// TIA Portal V20 export
FUNCTION_BLOCK "Sequence_10_GaugeRnR"   // FB32857, LAD
TITLE = Sequence
// Sequence template programmend in ladder logic
// stored: IsIECCheckEnabled true, MemoryReserve 100, Namespace Unit1.Em5, SetENOAutomatically true
   VAR_INPUT
      unitStatus { ExternalAccessible := 'False'; ExternalVisible := 'False'; ExternalWritable := 'False'} : "LAF_typeUnitStatus";
   END_VAR
   VAR
      instSequenceLADControl { ExternalWritable := 'False'} : "LAF_ControlLadSequence";
      instSequenceLADStatus { ExternalWritable := 'False'} : "LAF_StatusLadSequence";
      statTonTime { ExternalAccessible := 'False'; ExternalVisible := 'False'; ExternalWritable := 'False'} : Array[0..9999] of TON_TIME;
   END_VAR
   VAR_TEMP
      tempCustomerAction : Bool;   // Placeholder for possible actions
      tempDo_nothing_and_wait_for_init : Bool;   // Placeholder for doing nothing
      tempSafeStateCondition : Bool;   // Temp Condition for the equipment module to be in a safe state
   END_VAR
   VAR CONSTANT
      delayTime : Time := T#500ms;
      STEP_IDLE : DInt := 1;
      JOB_1_STEP_01 : DInt := 101;
      JOB_1_STEP_10 : DInt := 110;
      JOB_1_STEP_20 : DInt := 120;
      JOB_1_STEP_30 : DInt := 130;
      JOB_1_STEP_40 : DInt := 140;
      JOB_1_STEP_50 : DInt := 150;
      JOB_1_STEP_60 : DInt := 160;
      JOB_1_STEP_70 : DInt := 170;
      JOB_1_STEP_80 : DInt := 180;
      JOB_1_STEP_90 : DInt := 190;
      JOB_2_STEP_01 : DInt := 201;
      JOB_2_STEP_10 : DInt := 210;
      JOB_2_STEP_20 : DInt := 220;
      JOB_2_STEP_30 : DInt := 230;
      JOB_2_STEP_40 : DInt := 240;
      JOB_2_STEP_41 : DInt := 241;
      JOB_2_STEP_80 : DInt := 280;
      JOB_2_STEP_81 : DInt := 281;
      JOB_2_STEP_90 : DInt := 290;
      JOB_3_STEP_01 : DInt := 301;
      JOB_3_STEP_10 : DInt := 310;
      JOB_3_STEP_20 : DInt := 320;
      JOB_3_STEP_30 : DInt := 330;
      JOB_3_STEP_40 : DInt := 340;
      JOB_3_STEP_50 : DInt := 350;
      JOB_3_STEP_80 : DInt := 380;
      JOB_3_STEP_81 : DInt := 381;
      JOB_3_STEP_82 : DInt := 382;
      JOB_3_STEP_90 : DInt := 390;
      JOB_4_STEP_01 : DInt := 401;
      JOB_4_STEP_10 : DInt := 410;
      JOB_4_STEP_20 : DInt := 420;
      JOB_4_STEP_30 : DInt := 430;
      JOB_4_STEP_40 : DInt := 440;
      JOB_4_STEP_50 : DInt := 450;
      JOB_4_STEP_60 : DInt := 460;
      JOB_4_STEP_70 : DInt := 470;
      JOB_4_STEP_80 : DInt := 480;
      JOB_4_STEP_81 : DInt := 481;
      JOB_4_STEP_90 : DInt := 490;
      JOB_5_STEP_01 : DInt := 501;
      JOB_5_STEP_10 : DInt := 510;
      JOB_5_STEP_20 : DInt := 520;
      JOB_5_STEP_30 : DInt := 530;
      JOB_5_STEP_40 : DInt := 540;
      JOB_5_STEP_50 : DInt := 550;
      JOB_5_STEP_60 : DInt := 560;
      JOB_5_STEP_70 : DInt := 570;
      JOB_5_STEP_80 : DInt := 580;
      JOB_5_STEP_81 : DInt := 581;
      JOB_5_STEP_90 : DInt := 590;
      JOB_6_STEP_01 : DInt := 601;
      JOB_6_STEP_10 : DInt := 610;
      JOB_6_STEP_20 : DInt := 620;
      JOB_6_STEP_30 : DInt := 630;
      JOB_6_STEP_40 : DInt := 640;
      JOB_6_STEP_50 : DInt := 650;
      JOB_6_STEP_60 : DInt := 660;
      JOB_6_STEP_70 : DInt := 670;
      JOB_6_STEP_80 : DInt := 680;
      JOB_6_STEP_81 : DInt := 681;
      JOB_6_STEP_82 : DInt := 682;
      JOB_6_STEP_90 : DInt := 690;
      JOB_7_STEP_01 : DInt := 701;
      JOB_7_STEP_10 : DInt := 710;
      JOB_7_STEP_20 : DInt := 720;
      JOB_7_STEP_30 : DInt := 730;
      JOB_7_STEP_40 : DInt := 740;
      JOB_7_STEP_50 : DInt := 750;
      JOB_7_STEP_60 : DInt := 760;
      JOB_7_STEP_70 : DInt := 770;
      JOB_7_STEP_80 : DInt := 780;
      JOB_7_STEP_81 : DInt := 781;
      JOB_7_STEP_82 : DInt := 782;
      JOB_7_STEP_90 : DInt := 790;
      JOB_8_STEP_01 : DInt := 801;
      JOB_8_STEP_10 : DInt := 810;
      JOB_8_STEP_20 : DInt := 820;
      JOB_8_STEP_30 : DInt := 830;
      JOB_8_STEP_31 : DInt := 831;
      JOB_8_STEP_40 : DInt := 840;
      JOB_8_STEP_50 : DInt := 850;
      JOB_8_STEP_80 : DInt := 880;
      JOB_8_STEP_81 : DInt := 881;
      JOB_8_STEP_90 : DInt := 890;
      JOB_9_STEP_01 : DInt := 901;
      JOB_9_STEP_10 : DInt := 910;
      JOB_9_STEP_20 : DInt := 920;
      JOB_9_STEP_30 : DInt := 930;
      JOB_9_STEP_40 : DInt := 940;
      JOB_9_STEP_80 : DInt := 980;
      JOB_9_STEP_81 : DInt := 981;
      JOB_9_STEP_90 : DInt := 990;
      STEP_IMMEDIATE_STOP : DInt := 9001;   // Step executed when an immediate stop command is triggered for the sequence (i.e. when unit is in state aborting)
      TO_DO_INSERT_ACTIONS_HERE : Bool := TRUE;   // Template : Add actions
      TO_DO_INSERT_CONDITION_FOR_TRANSITION_HERE : Bool := TRUE;   // Template : Add conditions
   END_VAR
   VAR_TEMP   // added for the SCL form of the ladder/FBD networks
      _w1 : Bool;
   END_VAR
BEGIN

REGION Network 1: BLOCK INFO HEADER
   // (company) / (C) Copyright (year)
   // ---------------------------------------------------------------------------------
   // Title:                             (Title of this block)
   // Comment/Function: (that is implemented in the block)
   // Library/Family:           (that the source is dedicated to)
   // Author:                        (department / person in charge / contact)
   // Target System:          (test system with FW version)
   // Engineering:              TIA Portal (SW version)
   // Restrictions:               (OB types, etc.)
   // Requirements:           (hardware, technological package, etc.)
   // ---------------------------------------------------------------------------------
   // Change log table:
   // Version          | Date             | Signature      | Expert in charge  | Changes applied ------------------------|----------------------|-------------------------|--------------------------------|-----------------------
   // 001.000.000 | yyyy-mm-dd | 0x00000000 | (name of expert) | First released version
END_REGION

REGION Network 2: DESCRIPTION
   // This is a template block provided by the Automation Framework. It can be used to create an own project.
   // The Block Info Header is prepared to put in your own data.
   // Description of the block could be added here and the docu created by Code2Docu.
END_REGION

REGION Network 3: ********************* CONTROL *************************
END_REGION

REGION Network 4: Sequence Control ("Enter your Sequins number here")
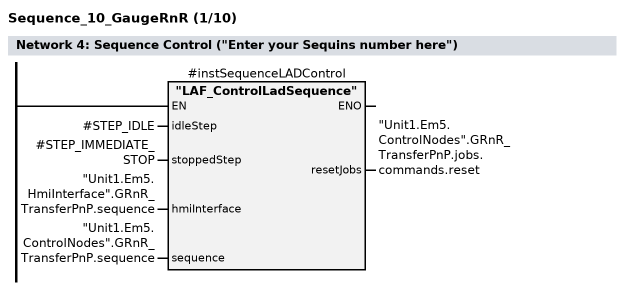
   RUNG wire#powerrail
      #instSequenceLADControl(idleStep := #STEP_IDLE, stoppedStep := #STEP_IMMEDIATE_STOP, hmiInterface := "Unit1.Em5.HmiInterface".GRnR_TransferPnP.sequence, sequence := "Unit1.Em5.ControlNodes".GRnR_TransferPnP.sequence, resetJobs => "Unit1.Em5.ControlNodes".GRnR_TransferPnP.jobs.commands.reset)
   END_RUNG
   // the same network as SCL:
   #instSequenceLADControl(idleStep := #STEP_IDLE,   // "LAF_ControlLadSequence"
                           stoppedStep := #STEP_IMMEDIATE_STOP,
                           hmiInterface := "Unit1.Em5.HmiInterface".GRnR_TransferPnP.sequence,
                           sequence := "Unit1.Em5.ControlNodes".GRnR_TransferPnP.sequence,
                           resetJobs => "Unit1.Em5.ControlNodes".GRnR_TransferPnP.jobs.commands.reset);
END_REGION

REGION Network 5: Step Idle
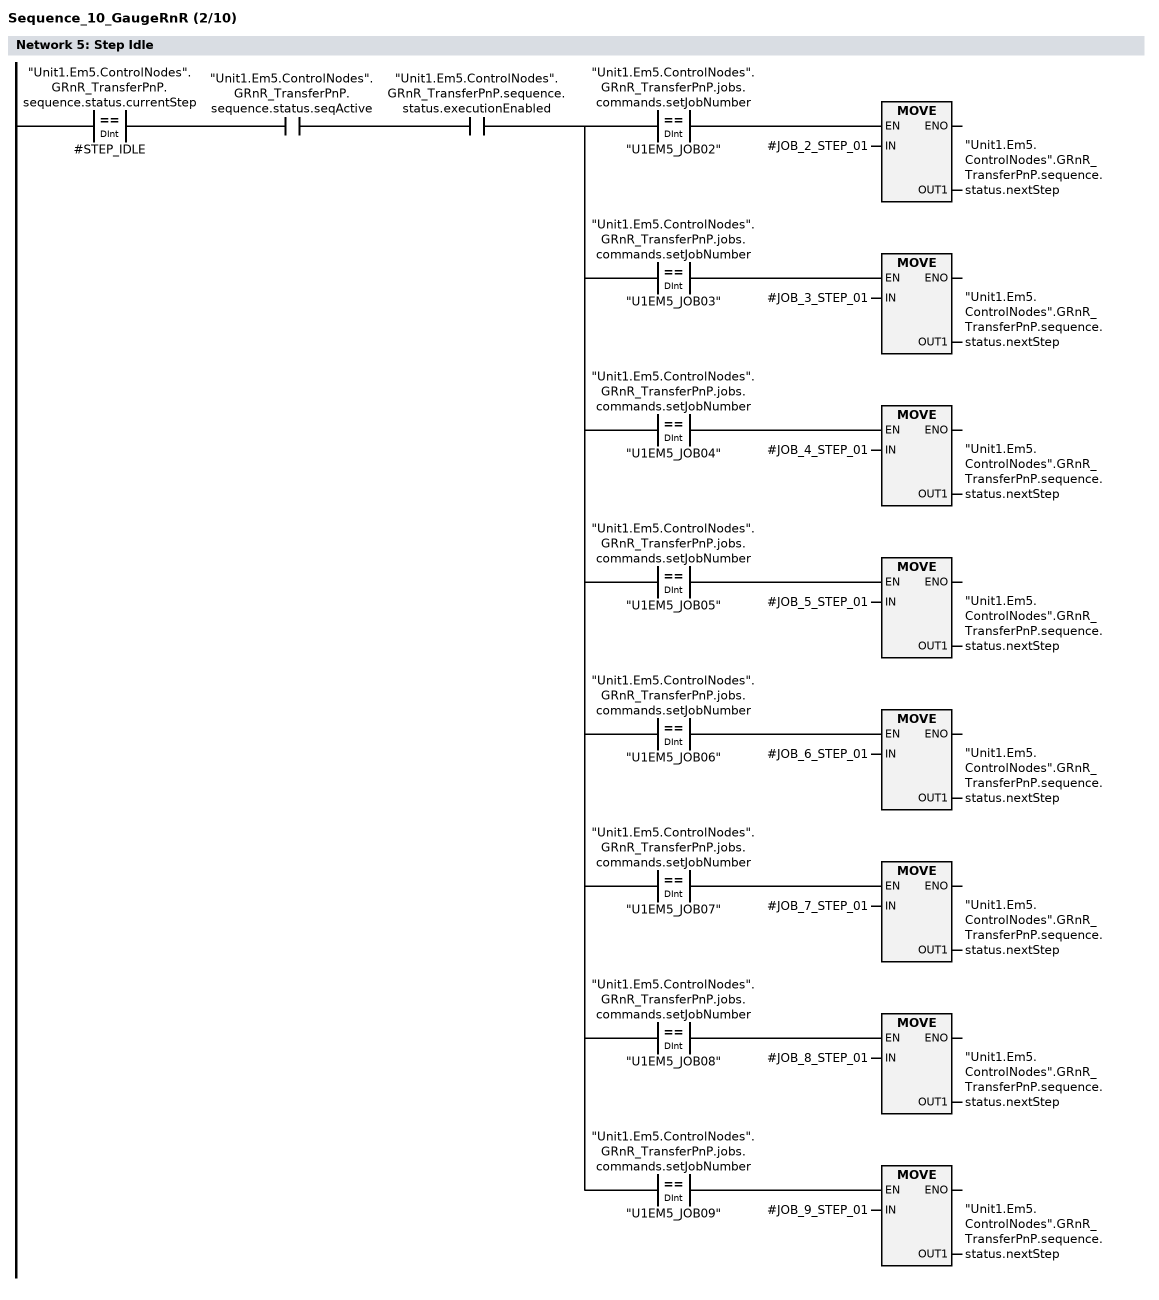
   RUNG wire#powerrail
      { S7_Templates := "SrcType := DInt" } EQ_Contact(in1 := "Unit1.Em5.ControlNodes".GRnR_TransferPnP.sequence.status.currentStep, in2 := #STEP_IDLE)
      Contact( "Unit1.Em5.ControlNodes".GRnR_TransferPnP.sequence.status.seqActive )
      Contact( "Unit1.Em5.ControlNodes".GRnR_TransferPnP.sequence.status.executionEnabled )
      wire#w1
      { S7_Templates := "SrcType := DInt" } EQ_Contact(in1 := "Unit1.Em5.ControlNodes".GRnR_TransferPnP.jobs.commands.setJobNumber, in2 := "U1EM5_JOB02")
      Move(in := #JOB_2_STEP_01, out1 => "Unit1.Em5.ControlNodes".GRnR_TransferPnP.sequence.status.nextStep)
   END_RUNG
   RUNG wire#w1
      { S7_Templates := "SrcType := DInt" } EQ_Contact(in1 := "Unit1.Em5.ControlNodes".GRnR_TransferPnP.jobs.commands.setJobNumber, in2 := "U1EM5_JOB03")
      Move(in := #JOB_3_STEP_01, out1 => "Unit1.Em5.ControlNodes".GRnR_TransferPnP.sequence.status.nextStep)
   END_RUNG
   RUNG wire#w1
      { S7_Templates := "SrcType := DInt" } EQ_Contact(in1 := "Unit1.Em5.ControlNodes".GRnR_TransferPnP.jobs.commands.setJobNumber, in2 := "U1EM5_JOB04")
      Move(in := #JOB_4_STEP_01, out1 => "Unit1.Em5.ControlNodes".GRnR_TransferPnP.sequence.status.nextStep)
   END_RUNG
   RUNG wire#w1
      { S7_Templates := "SrcType := DInt" } EQ_Contact(in1 := "Unit1.Em5.ControlNodes".GRnR_TransferPnP.jobs.commands.setJobNumber, in2 := "U1EM5_JOB05")
      Move(in := #JOB_5_STEP_01, out1 => "Unit1.Em5.ControlNodes".GRnR_TransferPnP.sequence.status.nextStep)
   END_RUNG
   RUNG wire#w1
      { S7_Templates := "SrcType := DInt" } EQ_Contact(in1 := "Unit1.Em5.ControlNodes".GRnR_TransferPnP.jobs.commands.setJobNumber, in2 := "U1EM5_JOB06")
      Move(in := #JOB_6_STEP_01, out1 => "Unit1.Em5.ControlNodes".GRnR_TransferPnP.sequence.status.nextStep)
   END_RUNG
   RUNG wire#w1
      { S7_Templates := "SrcType := DInt" } EQ_Contact(in1 := "Unit1.Em5.ControlNodes".GRnR_TransferPnP.jobs.commands.setJobNumber, in2 := "U1EM5_JOB07")
      Move(in := #JOB_7_STEP_01, out1 => "Unit1.Em5.ControlNodes".GRnR_TransferPnP.sequence.status.nextStep)
   END_RUNG
   RUNG wire#w1
      { S7_Templates := "SrcType := DInt" } EQ_Contact(in1 := "Unit1.Em5.ControlNodes".GRnR_TransferPnP.jobs.commands.setJobNumber, in2 := "U1EM5_JOB08")
      Move(in := #JOB_8_STEP_01, out1 => "Unit1.Em5.ControlNodes".GRnR_TransferPnP.sequence.status.nextStep)
   END_RUNG
   RUNG wire#w1
      { S7_Templates := "SrcType := DInt" } EQ_Contact(in1 := "Unit1.Em5.ControlNodes".GRnR_TransferPnP.jobs.commands.setJobNumber, in2 := "U1EM5_JOB09")
      Move(in := #JOB_9_STEP_01, out1 => "Unit1.Em5.ControlNodes".GRnR_TransferPnP.sequence.status.nextStep)
   END_RUNG
   // the same network as SCL:
   #_w1 := ("Unit1.Em5.ControlNodes".GRnR_TransferPnP.sequence.status.currentStep = #STEP_IDLE) AND "Unit1.Em5.ControlNodes".GRnR_TransferPnP.sequence.status.seqActive AND "Unit1.Em5.ControlNodes".GRnR_TransferPnP.sequence.status.executionEnabled;
   IF #_w1 AND ("Unit1.Em5.ControlNodes".GRnR_TransferPnP.jobs.commands.setJobNumber = "U1EM5_JOB02") THEN
       "Unit1.Em5.ControlNodes".GRnR_TransferPnP.sequence.status.nextStep := #JOB_2_STEP_01;
   END_IF;
   IF #_w1 AND ("Unit1.Em5.ControlNodes".GRnR_TransferPnP.jobs.commands.setJobNumber = "U1EM5_JOB03") THEN
       "Unit1.Em5.ControlNodes".GRnR_TransferPnP.sequence.status.nextStep := #JOB_3_STEP_01;
   END_IF;
   IF #_w1 AND ("Unit1.Em5.ControlNodes".GRnR_TransferPnP.jobs.commands.setJobNumber = "U1EM5_JOB04") THEN
       "Unit1.Em5.ControlNodes".GRnR_TransferPnP.sequence.status.nextStep := #JOB_4_STEP_01;
   END_IF;
   IF #_w1 AND ("Unit1.Em5.ControlNodes".GRnR_TransferPnP.jobs.commands.setJobNumber = "U1EM5_JOB05") THEN
       "Unit1.Em5.ControlNodes".GRnR_TransferPnP.sequence.status.nextStep := #JOB_5_STEP_01;
   END_IF;
   IF #_w1 AND ("Unit1.Em5.ControlNodes".GRnR_TransferPnP.jobs.commands.setJobNumber = "U1EM5_JOB06") THEN
       "Unit1.Em5.ControlNodes".GRnR_TransferPnP.sequence.status.nextStep := #JOB_6_STEP_01;
   END_IF;
   IF #_w1 AND ("Unit1.Em5.ControlNodes".GRnR_TransferPnP.jobs.commands.setJobNumber = "U1EM5_JOB07") THEN
       "Unit1.Em5.ControlNodes".GRnR_TransferPnP.sequence.status.nextStep := #JOB_7_STEP_01;
   END_IF;
   IF #_w1 AND ("Unit1.Em5.ControlNodes".GRnR_TransferPnP.jobs.commands.setJobNumber = "U1EM5_JOB08") THEN
       "Unit1.Em5.ControlNodes".GRnR_TransferPnP.sequence.status.nextStep := #JOB_8_STEP_01;
   END_IF;
   IF #_w1 AND ("Unit1.Em5.ControlNodes".GRnR_TransferPnP.jobs.commands.setJobNumber = "U1EM5_JOB09") THEN
       "Unit1.Em5.ControlNodes".GRnR_TransferPnP.sequence.status.nextStep := #JOB_9_STEP_01;
   END_IF;
END_REGION

REGION Network 6: *********** JOB[5] HIPOT & THICKNESS JR GET=R&R AUTO/TR RIGHT ************
END_REGION

REGION Network 7: Step[501] : JOB[5] Condition
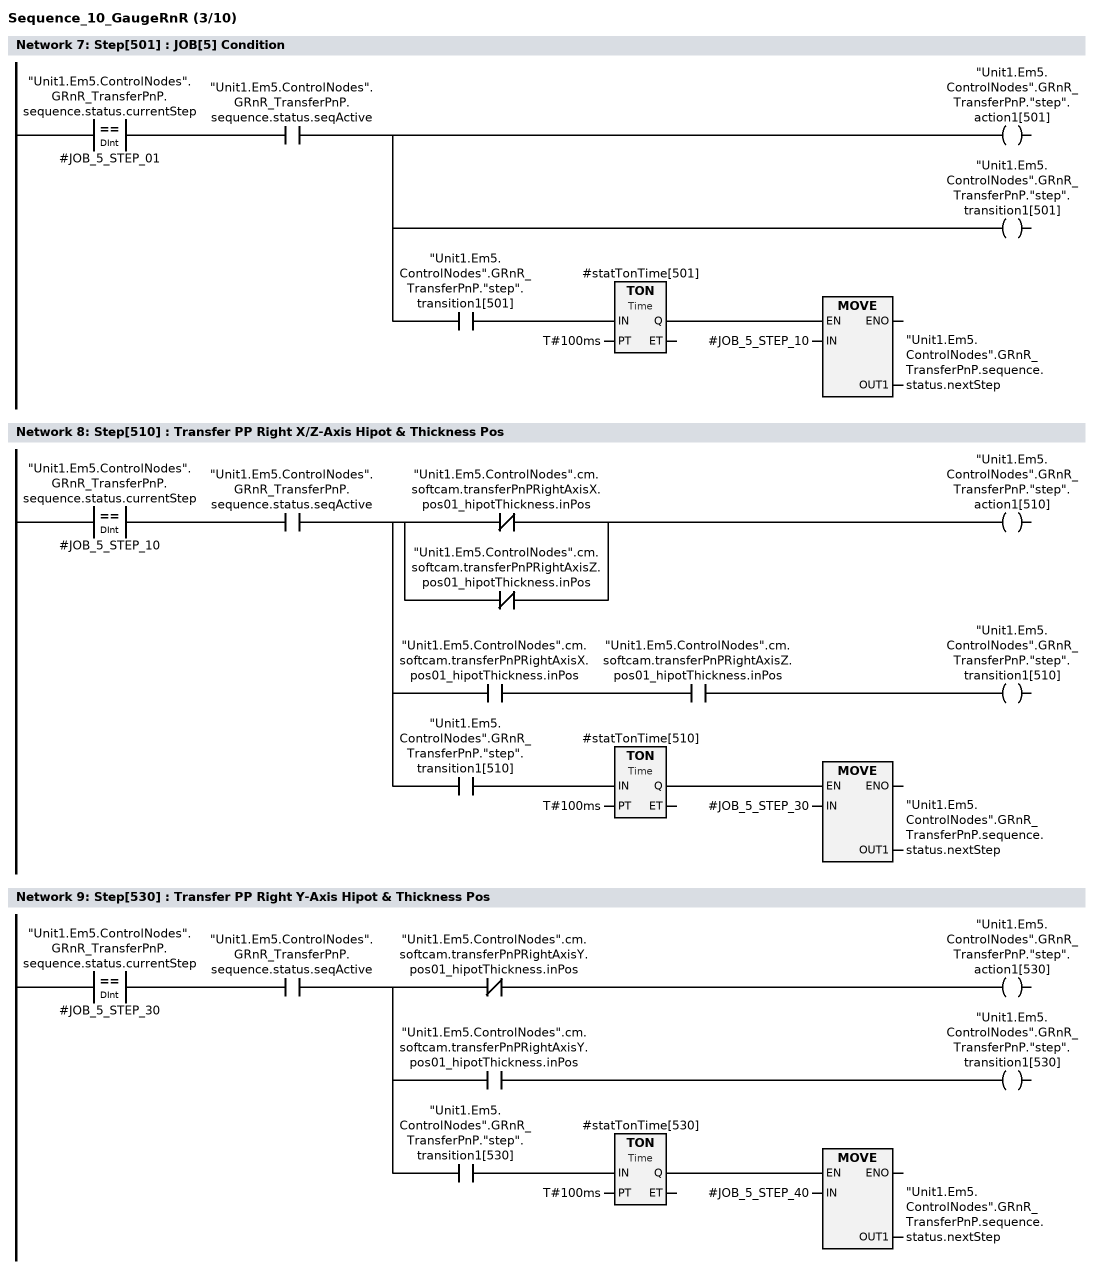
   RUNG wire#powerrail
      { S7_Templates := "SrcType := DInt" } EQ_Contact(in1 := "Unit1.Em5.ControlNodes".GRnR_TransferPnP.sequence.status.currentStep, in2 := #JOB_5_STEP_01)
      Contact( "Unit1.Em5.ControlNodes".GRnR_TransferPnP.sequence.status.seqActive )
      wire#w1
      Coil( "Unit1.Em5.ControlNodes".GRnR_TransferPnP."step".action1[501] )
   END_RUNG
   RUNG wire#w1
      Coil( "Unit1.Em5.ControlNodes".GRnR_TransferPnP."step".transition1[501] )
   END_RUNG
   RUNG wire#w1
      Contact( "Unit1.Em5.ControlNodes".GRnR_TransferPnP."step".transition1[501] )
      { S7_Templates := "time_type := Time" } #statTonTime[501].TON(pt := T#100ms, et =>)
      Move(in := #JOB_5_STEP_10, out1 => "Unit1.Em5.ControlNodes".GRnR_TransferPnP.sequence.status.nextStep)
   END_RUNG
   // the same network as SCL:
   "Unit1.Em5.ControlNodes".GRnR_TransferPnP."step".action1[501] := ("Unit1.Em5.ControlNodes".GRnR_TransferPnP.sequence.status.currentStep = #JOB_5_STEP_01) AND "Unit1.Em5.ControlNodes".GRnR_TransferPnP.sequence.status.seqActive;
   "Unit1.Em5.ControlNodes".GRnR_TransferPnP."step".transition1[501] := ("Unit1.Em5.ControlNodes".GRnR_TransferPnP.sequence.status.currentStep = #JOB_5_STEP_01) AND "Unit1.Em5.ControlNodes".GRnR_TransferPnP.sequence.status.seqActive;
   #statTonTime[501].TON(IN := ("Unit1.Em5.ControlNodes".GRnR_TransferPnP.sequence.status.currentStep = #JOB_5_STEP_01) AND "Unit1.Em5.ControlNodes".GRnR_TransferPnP.sequence.status.seqActive AND "Unit1.Em5.ControlNodes".GRnR_TransferPnP."step".transition1[501],
                         PT := T#100ms);
   IF #statTonTime[501].Q THEN
       "Unit1.Em5.ControlNodes".GRnR_TransferPnP.sequence.status.nextStep := #JOB_5_STEP_10;
   END_IF;
END_REGION

REGION Network 8: Step[510] : Transfer PP Right X/Z-Axis Hipot & Thickness Pos
   RUNG wire#powerrail
      { S7_Templates := "SrcType := DInt" } EQ_Contact(in1 := "Unit1.Em5.ControlNodes".GRnR_TransferPnP.sequence.status.currentStep, in2 := #JOB_5_STEP_10)
      Contact( "Unit1.Em5.ControlNodes".GRnR_TransferPnP.sequence.status.seqActive )
      wire#w1
      I_Contact( "Unit1.Em5.ControlNodes".cm.softcam.transferPnPRightAxisX.pos01_hipotThickness.inPos )
      wire#w2
      Coil( "Unit1.Em5.ControlNodes".GRnR_TransferPnP."step".action1[510] )
   END_RUNG
   RUNG wire#w1
      I_Contact( "Unit1.Em5.ControlNodes".cm.softcam.transferPnPRightAxisZ.pos01_hipotThickness.inPos )
   END_RUNG wire#w2
   RUNG wire#w1
      Contact( "Unit1.Em5.ControlNodes".cm.softcam.transferPnPRightAxisX.pos01_hipotThickness.inPos )
      Contact( "Unit1.Em5.ControlNodes".cm.softcam.transferPnPRightAxisZ.pos01_hipotThickness.inPos )
      Coil( "Unit1.Em5.ControlNodes".GRnR_TransferPnP."step".transition1[510] )
   END_RUNG
   RUNG wire#w1
      Contact( "Unit1.Em5.ControlNodes".GRnR_TransferPnP."step".transition1[510] )
      { S7_Templates := "time_type := Time" } #statTonTime[510].TON(pt := T#100ms, et =>)
      Move(in := #JOB_5_STEP_30, out1 => "Unit1.Em5.ControlNodes".GRnR_TransferPnP.sequence.status.nextStep)
   END_RUNG
   // the same network as SCL:
   #_w1 := ("Unit1.Em5.ControlNodes".GRnR_TransferPnP.sequence.status.currentStep = #JOB_5_STEP_10) AND "Unit1.Em5.ControlNodes".GRnR_TransferPnP.sequence.status.seqActive;
   "Unit1.Em5.ControlNodes".GRnR_TransferPnP."step".action1[510] := #_w1 AND (NOT "Unit1.Em5.ControlNodes".cm.softcam.transferPnPRightAxisX.pos01_hipotThickness.inPos OR NOT "Unit1.Em5.ControlNodes".cm.softcam.transferPnPRightAxisZ.pos01_hipotThickness.inPos);
   "Unit1.Em5.ControlNodes".GRnR_TransferPnP."step".transition1[510] := #_w1 AND "Unit1.Em5.ControlNodes".cm.softcam.transferPnPRightAxisX.pos01_hipotThickness.inPos AND "Unit1.Em5.ControlNodes".cm.softcam.transferPnPRightAxisZ.pos01_hipotThickness.inPos;
   #statTonTime[510].TON(IN := #_w1 AND "Unit1.Em5.ControlNodes".GRnR_TransferPnP."step".transition1[510],
                         PT := T#100ms);
   IF #statTonTime[510].Q THEN
       "Unit1.Em5.ControlNodes".GRnR_TransferPnP.sequence.status.nextStep := #JOB_5_STEP_30;
   END_IF;
END_REGION

REGION Network 9: Step[530] : Transfer PP Right Y-Axis Hipot & Thickness Pos
   RUNG wire#powerrail
      { S7_Templates := "SrcType := DInt" } EQ_Contact(in1 := "Unit1.Em5.ControlNodes".GRnR_TransferPnP.sequence.status.currentStep, in2 := #JOB_5_STEP_30)
      Contact( "Unit1.Em5.ControlNodes".GRnR_TransferPnP.sequence.status.seqActive )
      wire#w1
      I_Contact( "Unit1.Em5.ControlNodes".cm.softcam.transferPnPRightAxisY.pos01_hipotThickness.inPos )
      Coil( "Unit1.Em5.ControlNodes".GRnR_TransferPnP."step".action1[530] )
   END_RUNG
   RUNG wire#w1
      Contact( "Unit1.Em5.ControlNodes".cm.softcam.transferPnPRightAxisY.pos01_hipotThickness.inPos )
      Coil( "Unit1.Em5.ControlNodes".GRnR_TransferPnP."step".transition1[530] )
   END_RUNG
   RUNG wire#w1
      Contact( "Unit1.Em5.ControlNodes".GRnR_TransferPnP."step".transition1[530] )
      { S7_Templates := "time_type := Time" } #statTonTime[530].TON(pt := T#100ms, et =>)
      Move(in := #JOB_5_STEP_40, out1 => "Unit1.Em5.ControlNodes".GRnR_TransferPnP.sequence.status.nextStep)
   END_RUNG
   // the same network as SCL:
   #_w1 := ("Unit1.Em5.ControlNodes".GRnR_TransferPnP.sequence.status.currentStep = #JOB_5_STEP_30) AND "Unit1.Em5.ControlNodes".GRnR_TransferPnP.sequence.status.seqActive;
   "Unit1.Em5.ControlNodes".GRnR_TransferPnP."step".action1[530] := #_w1 AND NOT "Unit1.Em5.ControlNodes".cm.softcam.transferPnPRightAxisY.pos01_hipotThickness.inPos;
   "Unit1.Em5.ControlNodes".GRnR_TransferPnP."step".transition1[530] := #_w1 AND "Unit1.Em5.ControlNodes".cm.softcam.transferPnPRightAxisY.pos01_hipotThickness.inPos;
   #statTonTime[530].TON(IN := #_w1 AND "Unit1.Em5.ControlNodes".GRnR_TransferPnP."step".transition1[530],
                         PT := T#100ms);
   IF #statTonTime[530].Q THEN
       "Unit1.Em5.ControlNodes".GRnR_TransferPnP.sequence.status.nextStep := #JOB_5_STEP_40;
   END_IF;
END_REGION

REGION Network 10: Step[540] : Transfer PP Right Clamp Close
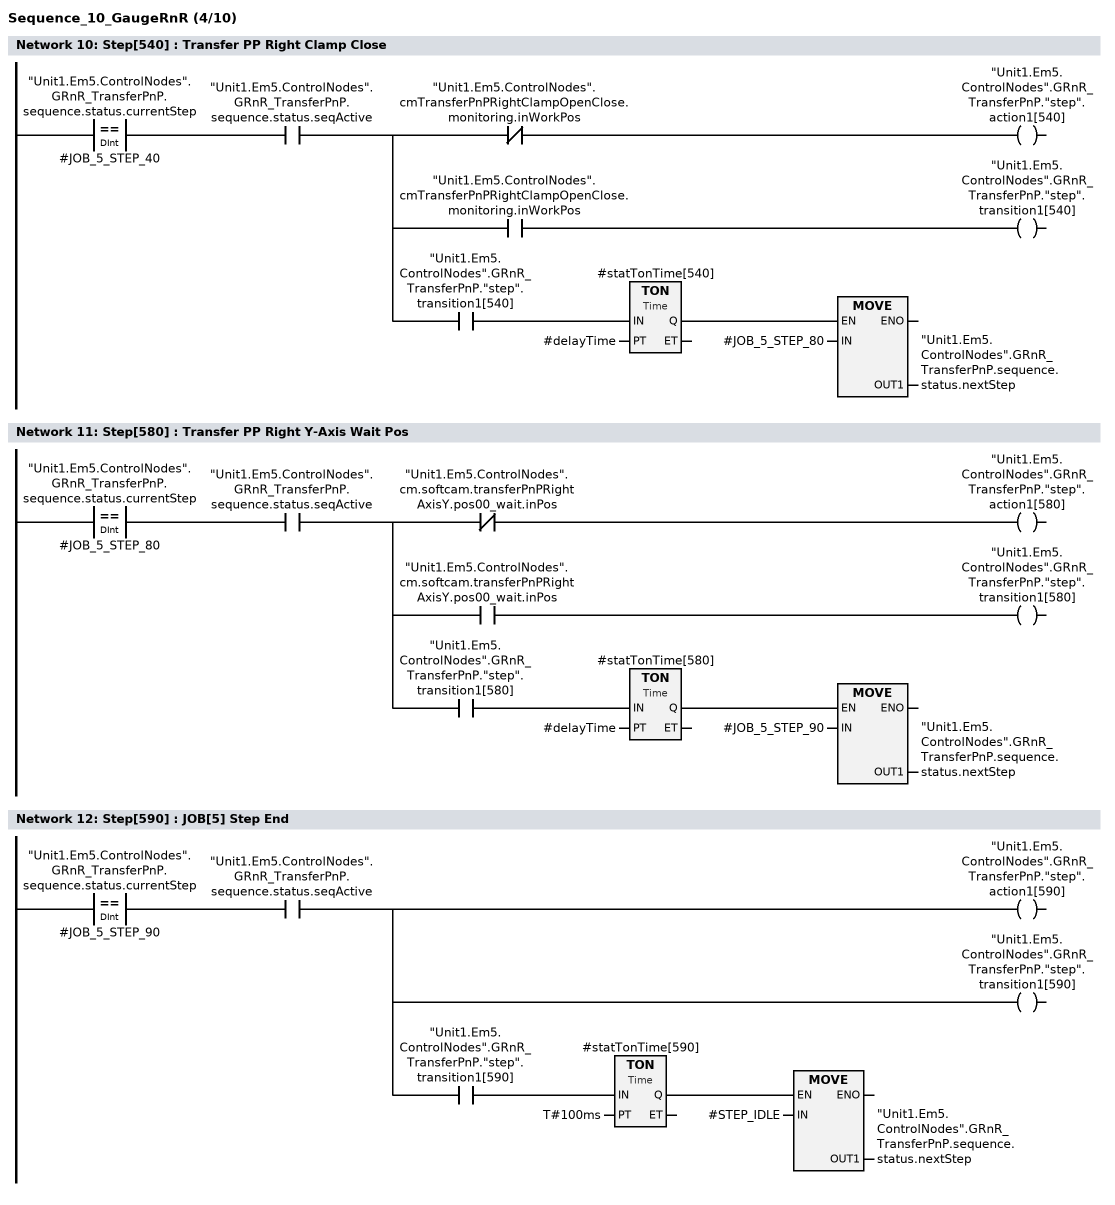
   RUNG wire#powerrail
      { S7_Templates := "SrcType := DInt" } EQ_Contact(in1 := "Unit1.Em5.ControlNodes".GRnR_TransferPnP.sequence.status.currentStep, in2 := #JOB_5_STEP_40)
      Contact( "Unit1.Em5.ControlNodes".GRnR_TransferPnP.sequence.status.seqActive )
      wire#w1
      I_Contact( "Unit1.Em5.ControlNodes".cmTransferPnPRightClampOpenClose.monitoring.inWorkPos )
      Coil( "Unit1.Em5.ControlNodes".GRnR_TransferPnP."step".action1[540] )
   END_RUNG
   RUNG wire#w1
      Contact( "Unit1.Em5.ControlNodes".cmTransferPnPRightClampOpenClose.monitoring.inWorkPos )
      Coil( "Unit1.Em5.ControlNodes".GRnR_TransferPnP."step".transition1[540] )
   END_RUNG
   RUNG wire#w1
      Contact( "Unit1.Em5.ControlNodes".GRnR_TransferPnP."step".transition1[540] )
      { S7_Templates := "time_type := Time" } #statTonTime[540].TON(pt := #delayTime, et =>)
      Move(in := #JOB_5_STEP_80, out1 => "Unit1.Em5.ControlNodes".GRnR_TransferPnP.sequence.status.nextStep)
   END_RUNG
   // the same network as SCL:
   #_w1 := ("Unit1.Em5.ControlNodes".GRnR_TransferPnP.sequence.status.currentStep = #JOB_5_STEP_40) AND "Unit1.Em5.ControlNodes".GRnR_TransferPnP.sequence.status.seqActive;
   "Unit1.Em5.ControlNodes".GRnR_TransferPnP."step".action1[540] := #_w1 AND NOT "Unit1.Em5.ControlNodes".cmTransferPnPRightClampOpenClose.monitoring.inWorkPos;
   "Unit1.Em5.ControlNodes".GRnR_TransferPnP."step".transition1[540] := #_w1 AND "Unit1.Em5.ControlNodes".cmTransferPnPRightClampOpenClose.monitoring.inWorkPos;
   #statTonTime[540].TON(IN := #_w1 AND "Unit1.Em5.ControlNodes".GRnR_TransferPnP."step".transition1[540],
                         PT := #delayTime);
   IF #statTonTime[540].Q THEN
       "Unit1.Em5.ControlNodes".GRnR_TransferPnP.sequence.status.nextStep := #JOB_5_STEP_80;
   END_IF;
END_REGION

REGION Network 11: Step[580] : Transfer PP Right Y-Axis Wait Pos
   RUNG wire#powerrail
      { S7_Templates := "SrcType := DInt" } EQ_Contact(in1 := "Unit1.Em5.ControlNodes".GRnR_TransferPnP.sequence.status.currentStep, in2 := #JOB_5_STEP_80)
      Contact( "Unit1.Em5.ControlNodes".GRnR_TransferPnP.sequence.status.seqActive )
      wire#w1
      I_Contact( "Unit1.Em5.ControlNodes".cm.softcam.transferPnPRightAxisY.pos00_wait.inPos )
      Coil( "Unit1.Em5.ControlNodes".GRnR_TransferPnP."step".action1[580] )
   END_RUNG
   RUNG wire#w1
      Contact( "Unit1.Em5.ControlNodes".cm.softcam.transferPnPRightAxisY.pos00_wait.inPos )
      Coil( "Unit1.Em5.ControlNodes".GRnR_TransferPnP."step".transition1[580] )
   END_RUNG
   RUNG wire#w1
      Contact( "Unit1.Em5.ControlNodes".GRnR_TransferPnP."step".transition1[580] )
      { S7_Templates := "time_type := Time" } #statTonTime[580].TON(pt := #delayTime, et =>)
      Move(in := #JOB_5_STEP_90, out1 => "Unit1.Em5.ControlNodes".GRnR_TransferPnP.sequence.status.nextStep)
   END_RUNG
   // the same network as SCL:
   #_w1 := ("Unit1.Em5.ControlNodes".GRnR_TransferPnP.sequence.status.currentStep = #JOB_5_STEP_80) AND "Unit1.Em5.ControlNodes".GRnR_TransferPnP.sequence.status.seqActive;
   "Unit1.Em5.ControlNodes".GRnR_TransferPnP."step".action1[580] := #_w1 AND NOT "Unit1.Em5.ControlNodes".cm.softcam.transferPnPRightAxisY.pos00_wait.inPos;
   "Unit1.Em5.ControlNodes".GRnR_TransferPnP."step".transition1[580] := #_w1 AND "Unit1.Em5.ControlNodes".cm.softcam.transferPnPRightAxisY.pos00_wait.inPos;
   #statTonTime[580].TON(IN := #_w1 AND "Unit1.Em5.ControlNodes".GRnR_TransferPnP."step".transition1[580],
                         PT := #delayTime);
   IF #statTonTime[580].Q THEN
       "Unit1.Em5.ControlNodes".GRnR_TransferPnP.sequence.status.nextStep := #JOB_5_STEP_90;
   END_IF;
END_REGION

REGION Network 12: Step[590] : JOB[5] Step End
   RUNG wire#powerrail
      { S7_Templates := "SrcType := DInt" } EQ_Contact(in1 := "Unit1.Em5.ControlNodes".GRnR_TransferPnP.sequence.status.currentStep, in2 := #JOB_5_STEP_90)
      Contact( "Unit1.Em5.ControlNodes".GRnR_TransferPnP.sequence.status.seqActive )
      wire#w1
      Coil( "Unit1.Em5.ControlNodes".GRnR_TransferPnP."step".action1[590] )
   END_RUNG
   RUNG wire#w1
      Coil( "Unit1.Em5.ControlNodes".GRnR_TransferPnP."step".transition1[590] )
   END_RUNG
   RUNG wire#w1
      Contact( "Unit1.Em5.ControlNodes".GRnR_TransferPnP."step".transition1[590] )
      { S7_Templates := "time_type := Time" } #statTonTime[590].TON(pt := T#100ms, et =>)
      Move(in := #STEP_IDLE, out1 => "Unit1.Em5.ControlNodes".GRnR_TransferPnP.sequence.status.nextStep)
   END_RUNG
   // the same network as SCL:
   "Unit1.Em5.ControlNodes".GRnR_TransferPnP."step".action1[590] := ("Unit1.Em5.ControlNodes".GRnR_TransferPnP.sequence.status.currentStep = #JOB_5_STEP_90) AND "Unit1.Em5.ControlNodes".GRnR_TransferPnP.sequence.status.seqActive;
   "Unit1.Em5.ControlNodes".GRnR_TransferPnP."step".transition1[590] := ("Unit1.Em5.ControlNodes".GRnR_TransferPnP.sequence.status.currentStep = #JOB_5_STEP_90) AND "Unit1.Em5.ControlNodes".GRnR_TransferPnP.sequence.status.seqActive;
   #statTonTime[590].TON(IN := ("Unit1.Em5.ControlNodes".GRnR_TransferPnP.sequence.status.currentStep = #JOB_5_STEP_90) AND "Unit1.Em5.ControlNodes".GRnR_TransferPnP.sequence.status.seqActive AND "Unit1.Em5.ControlNodes".GRnR_TransferPnP."step".transition1[590],
                         PT := T#100ms);
   IF #statTonTime[590].Q THEN
       "Unit1.Em5.ControlNodes".GRnR_TransferPnP.sequence.status.nextStep := #STEP_IDLE;
   END_IF;
END_REGION

REGION Network 13: **************** JOB[6] VISION JR PUT=R&R AUTO/TR RIGHT *****************
END_REGION

REGION Network 14: Step[601] : JOB[6] Condition
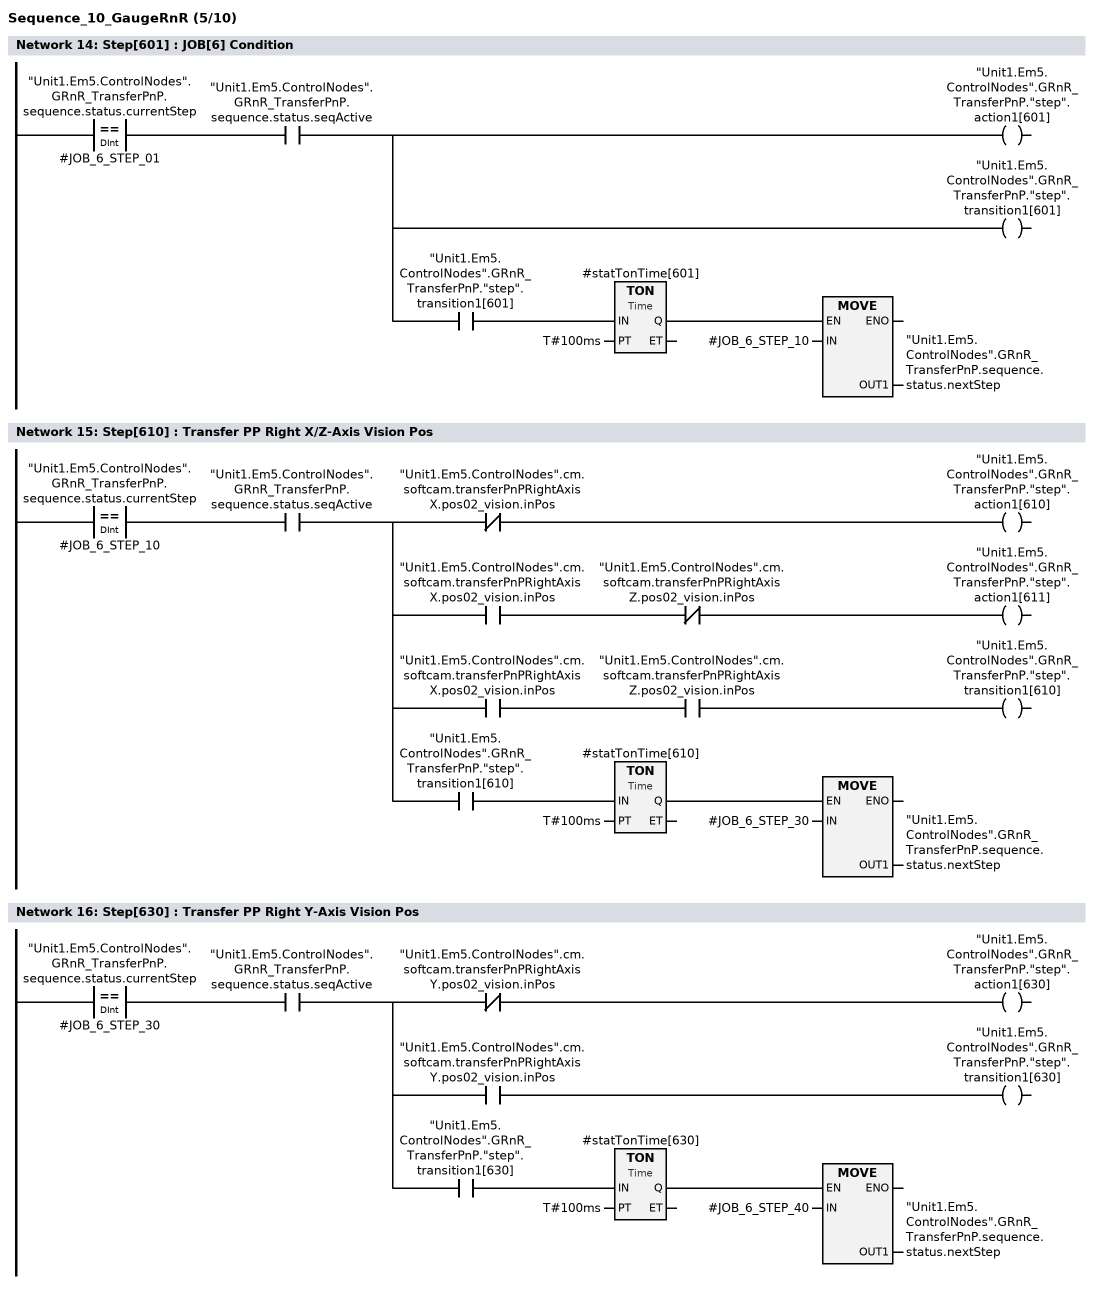
   RUNG wire#powerrail
      { S7_Templates := "SrcType := DInt" } EQ_Contact(in1 := "Unit1.Em5.ControlNodes".GRnR_TransferPnP.sequence.status.currentStep, in2 := #JOB_6_STEP_01)
      Contact( "Unit1.Em5.ControlNodes".GRnR_TransferPnP.sequence.status.seqActive )
      wire#w1
      Coil( "Unit1.Em5.ControlNodes".GRnR_TransferPnP."step".action1[601] )
   END_RUNG
   RUNG wire#w1
      Coil( "Unit1.Em5.ControlNodes".GRnR_TransferPnP."step".transition1[601] )
   END_RUNG
   RUNG wire#w1
      Contact( "Unit1.Em5.ControlNodes".GRnR_TransferPnP."step".transition1[601] )
      { S7_Templates := "time_type := Time" } #statTonTime[601].TON(pt := T#100ms, et =>)
      Move(in := #JOB_6_STEP_10, out1 => "Unit1.Em5.ControlNodes".GRnR_TransferPnP.sequence.status.nextStep)
   END_RUNG
   // the same network as SCL:
   "Unit1.Em5.ControlNodes".GRnR_TransferPnP."step".action1[601] := ("Unit1.Em5.ControlNodes".GRnR_TransferPnP.sequence.status.currentStep = #JOB_6_STEP_01) AND "Unit1.Em5.ControlNodes".GRnR_TransferPnP.sequence.status.seqActive;
   "Unit1.Em5.ControlNodes".GRnR_TransferPnP."step".transition1[601] := ("Unit1.Em5.ControlNodes".GRnR_TransferPnP.sequence.status.currentStep = #JOB_6_STEP_01) AND "Unit1.Em5.ControlNodes".GRnR_TransferPnP.sequence.status.seqActive;
   #statTonTime[601].TON(IN := ("Unit1.Em5.ControlNodes".GRnR_TransferPnP.sequence.status.currentStep = #JOB_6_STEP_01) AND "Unit1.Em5.ControlNodes".GRnR_TransferPnP.sequence.status.seqActive AND "Unit1.Em5.ControlNodes".GRnR_TransferPnP."step".transition1[601],
                         PT := T#100ms);
   IF #statTonTime[601].Q THEN
       "Unit1.Em5.ControlNodes".GRnR_TransferPnP.sequence.status.nextStep := #JOB_6_STEP_10;
   END_IF;
END_REGION

REGION Network 15: Step[610] : Transfer PP Right X/Z-Axis Vision Pos
   RUNG wire#powerrail
      { S7_Templates := "SrcType := DInt" } EQ_Contact(in1 := "Unit1.Em5.ControlNodes".GRnR_TransferPnP.sequence.status.currentStep, in2 := #JOB_6_STEP_10)
      Contact( "Unit1.Em5.ControlNodes".GRnR_TransferPnP.sequence.status.seqActive )
      wire#w1
      I_Contact( "Unit1.Em5.ControlNodes".cm.softcam.transferPnPRightAxisX.pos02_vision.inPos )
      Coil( "Unit1.Em5.ControlNodes".GRnR_TransferPnP."step".action1[610] )
   END_RUNG
   RUNG wire#w1
      Contact( "Unit1.Em5.ControlNodes".cm.softcam.transferPnPRightAxisX.pos02_vision.inPos )
      I_Contact( "Unit1.Em5.ControlNodes".cm.softcam.transferPnPRightAxisZ.pos02_vision.inPos )
      Coil( "Unit1.Em5.ControlNodes".GRnR_TransferPnP."step".action1[611] )
   END_RUNG
   RUNG wire#w1
      Contact( "Unit1.Em5.ControlNodes".cm.softcam.transferPnPRightAxisX.pos02_vision.inPos )
      Contact( "Unit1.Em5.ControlNodes".cm.softcam.transferPnPRightAxisZ.pos02_vision.inPos )
      Coil( "Unit1.Em5.ControlNodes".GRnR_TransferPnP."step".transition1[610] )
   END_RUNG
   RUNG wire#w1
      Contact( "Unit1.Em5.ControlNodes".GRnR_TransferPnP."step".transition1[610] )
      { S7_Templates := "time_type := Time" } #statTonTime[610].TON(pt := T#100ms, et =>)
      Move(in := #JOB_6_STEP_30, out1 => "Unit1.Em5.ControlNodes".GRnR_TransferPnP.sequence.status.nextStep)
   END_RUNG
   // the same network as SCL:
   #_w1 := ("Unit1.Em5.ControlNodes".GRnR_TransferPnP.sequence.status.currentStep = #JOB_6_STEP_10) AND "Unit1.Em5.ControlNodes".GRnR_TransferPnP.sequence.status.seqActive;
   "Unit1.Em5.ControlNodes".GRnR_TransferPnP."step".action1[610] := #_w1 AND NOT "Unit1.Em5.ControlNodes".cm.softcam.transferPnPRightAxisX.pos02_vision.inPos;
   "Unit1.Em5.ControlNodes".GRnR_TransferPnP."step".action1[611] := #_w1 AND "Unit1.Em5.ControlNodes".cm.softcam.transferPnPRightAxisX.pos02_vision.inPos AND NOT "Unit1.Em5.ControlNodes".cm.softcam.transferPnPRightAxisZ.pos02_vision.inPos;
   "Unit1.Em5.ControlNodes".GRnR_TransferPnP."step".transition1[610] := #_w1 AND "Unit1.Em5.ControlNodes".cm.softcam.transferPnPRightAxisX.pos02_vision.inPos AND "Unit1.Em5.ControlNodes".cm.softcam.transferPnPRightAxisZ.pos02_vision.inPos;
   #statTonTime[610].TON(IN := #_w1 AND "Unit1.Em5.ControlNodes".GRnR_TransferPnP."step".transition1[610],
                         PT := T#100ms);
   IF #statTonTime[610].Q THEN
       "Unit1.Em5.ControlNodes".GRnR_TransferPnP.sequence.status.nextStep := #JOB_6_STEP_30;
   END_IF;
END_REGION

REGION Network 16: Step[630] : Transfer PP Right Y-Axis Vision Pos
   RUNG wire#powerrail
      { S7_Templates := "SrcType := DInt" } EQ_Contact(in1 := "Unit1.Em5.ControlNodes".GRnR_TransferPnP.sequence.status.currentStep, in2 := #JOB_6_STEP_30)
      Contact( "Unit1.Em5.ControlNodes".GRnR_TransferPnP.sequence.status.seqActive )
      wire#w1
      I_Contact( "Unit1.Em5.ControlNodes".cm.softcam.transferPnPRightAxisY.pos02_vision.inPos )
      Coil( "Unit1.Em5.ControlNodes".GRnR_TransferPnP."step".action1[630] )
   END_RUNG
   RUNG wire#w1
      Contact( "Unit1.Em5.ControlNodes".cm.softcam.transferPnPRightAxisY.pos02_vision.inPos )
      Coil( "Unit1.Em5.ControlNodes".GRnR_TransferPnP."step".transition1[630] )
   END_RUNG
   RUNG wire#w1
      Contact( "Unit1.Em5.ControlNodes".GRnR_TransferPnP."step".transition1[630] )
      { S7_Templates := "time_type := Time" } #statTonTime[630].TON(pt := T#100ms, et =>)
      Move(in := #JOB_6_STEP_40, out1 => "Unit1.Em5.ControlNodes".GRnR_TransferPnP.sequence.status.nextStep)
   END_RUNG
   // the same network as SCL:
   #_w1 := ("Unit1.Em5.ControlNodes".GRnR_TransferPnP.sequence.status.currentStep = #JOB_6_STEP_30) AND "Unit1.Em5.ControlNodes".GRnR_TransferPnP.sequence.status.seqActive;
   "Unit1.Em5.ControlNodes".GRnR_TransferPnP."step".action1[630] := #_w1 AND NOT "Unit1.Em5.ControlNodes".cm.softcam.transferPnPRightAxisY.pos02_vision.inPos;
   "Unit1.Em5.ControlNodes".GRnR_TransferPnP."step".transition1[630] := #_w1 AND "Unit1.Em5.ControlNodes".cm.softcam.transferPnPRightAxisY.pos02_vision.inPos;
   #statTonTime[630].TON(IN := #_w1 AND "Unit1.Em5.ControlNodes".GRnR_TransferPnP."step".transition1[630],
                         PT := T#100ms);
   IF #statTonTime[630].Q THEN
       "Unit1.Em5.ControlNodes".GRnR_TransferPnP.sequence.status.nextStep := #JOB_6_STEP_40;
   END_IF;
END_REGION

REGION Network 17: Step[650] : Transfer PP Right [Lift Up Request] => Vision Check
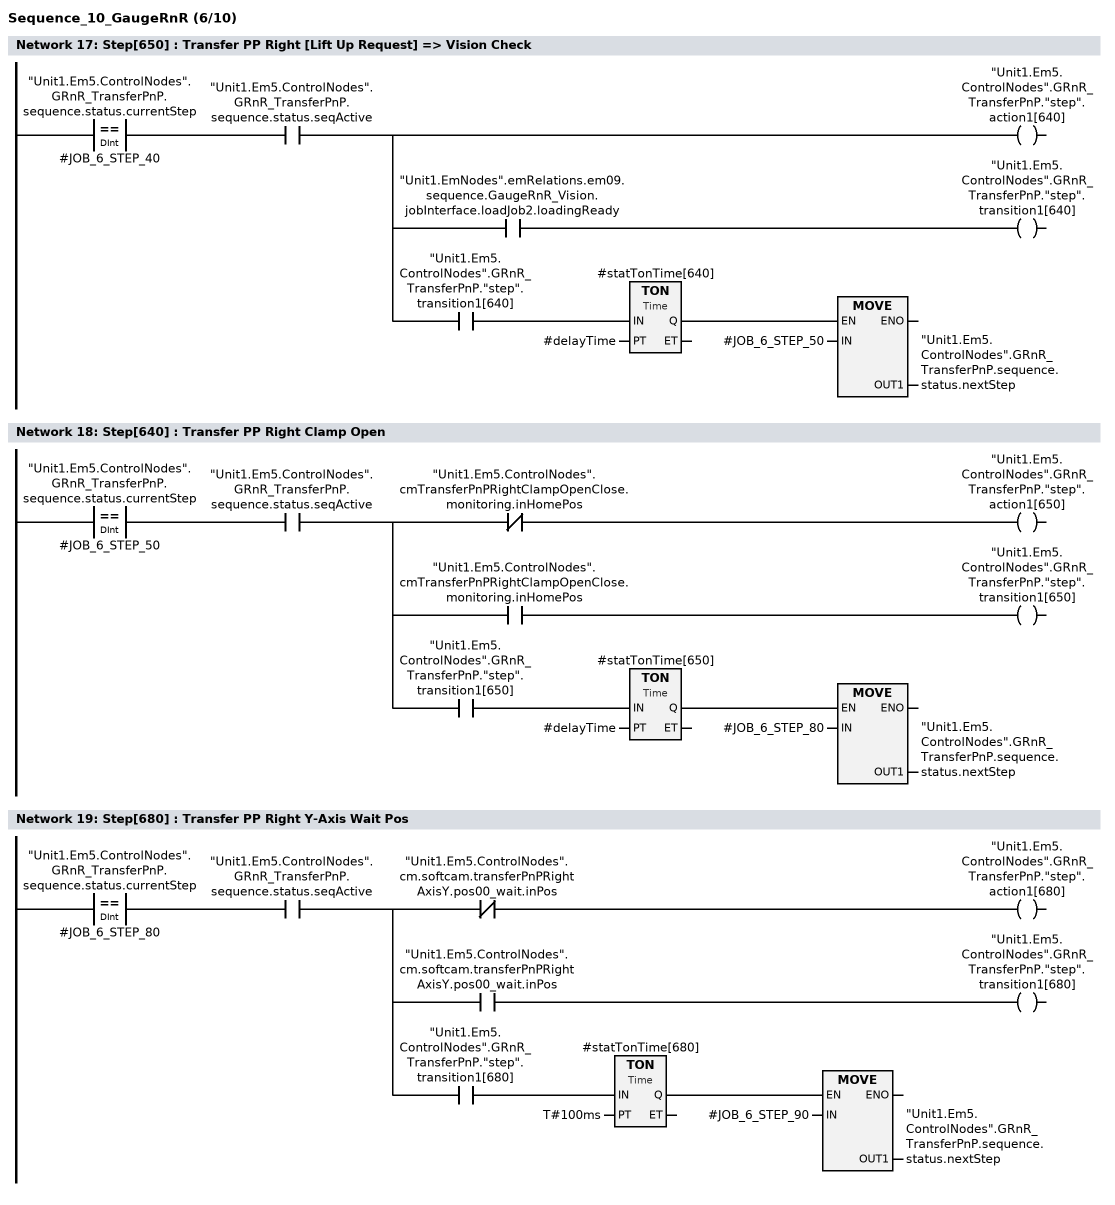
   RUNG wire#powerrail
      { S7_Templates := "SrcType := DInt" } EQ_Contact(in1 := "Unit1.Em5.ControlNodes".GRnR_TransferPnP.sequence.status.currentStep, in2 := #JOB_6_STEP_40)
      Contact( "Unit1.Em5.ControlNodes".GRnR_TransferPnP.sequence.status.seqActive )
      wire#w1
      Coil( "Unit1.Em5.ControlNodes".GRnR_TransferPnP."step".action1[640] )
   END_RUNG
   RUNG wire#w1
      Contact( "Unit1.EmNodes".emRelations.em09.sequence.GaugeRnR_Vision.jobInterface.loadJob2.loadingReady )
      Coil( "Unit1.Em5.ControlNodes".GRnR_TransferPnP."step".transition1[640] )
   END_RUNG
   RUNG wire#w1
      Contact( "Unit1.Em5.ControlNodes".GRnR_TransferPnP."step".transition1[640] )
      { S7_Templates := "time_type := Time" } #statTonTime[640].TON(pt := #delayTime, et =>)
      Move(in := #JOB_6_STEP_50, out1 => "Unit1.Em5.ControlNodes".GRnR_TransferPnP.sequence.status.nextStep)
   END_RUNG
   // the same network as SCL:
   "Unit1.Em5.ControlNodes".GRnR_TransferPnP."step".action1[640] := ("Unit1.Em5.ControlNodes".GRnR_TransferPnP.sequence.status.currentStep = #JOB_6_STEP_40) AND "Unit1.Em5.ControlNodes".GRnR_TransferPnP.sequence.status.seqActive;
   "Unit1.Em5.ControlNodes".GRnR_TransferPnP."step".transition1[640] := ("Unit1.Em5.ControlNodes".GRnR_TransferPnP.sequence.status.currentStep = #JOB_6_STEP_40) AND "Unit1.Em5.ControlNodes".GRnR_TransferPnP.sequence.status.seqActive AND "Unit1.EmNodes".emRelations.em09.sequence.GaugeRnR_Vision.jobInterface.loadJob2.loadingReady;
   #statTonTime[640].TON(IN := ("Unit1.Em5.ControlNodes".GRnR_TransferPnP.sequence.status.currentStep = #JOB_6_STEP_40) AND "Unit1.Em5.ControlNodes".GRnR_TransferPnP.sequence.status.seqActive AND "Unit1.Em5.ControlNodes".GRnR_TransferPnP."step".transition1[640],
                         PT := #delayTime);
   IF #statTonTime[640].Q THEN
       "Unit1.Em5.ControlNodes".GRnR_TransferPnP.sequence.status.nextStep := #JOB_6_STEP_50;
   END_IF;
END_REGION

REGION Network 18: Step[640] : Transfer PP Right Clamp Open
   RUNG wire#powerrail
      { S7_Templates := "SrcType := DInt" } EQ_Contact(in1 := "Unit1.Em5.ControlNodes".GRnR_TransferPnP.sequence.status.currentStep, in2 := #JOB_6_STEP_50)
      Contact( "Unit1.Em5.ControlNodes".GRnR_TransferPnP.sequence.status.seqActive )
      wire#w1
      I_Contact( "Unit1.Em5.ControlNodes".cmTransferPnPRightClampOpenClose.monitoring.inHomePos )
      Coil( "Unit1.Em5.ControlNodes".GRnR_TransferPnP."step".action1[650] )
   END_RUNG
   RUNG wire#w1
      Contact( "Unit1.Em5.ControlNodes".cmTransferPnPRightClampOpenClose.monitoring.inHomePos )
      Coil( "Unit1.Em5.ControlNodes".GRnR_TransferPnP."step".transition1[650] )
   END_RUNG
   RUNG wire#w1
      Contact( "Unit1.Em5.ControlNodes".GRnR_TransferPnP."step".transition1[650] )
      { S7_Templates := "time_type := Time" } #statTonTime[650].TON(pt := #delayTime, et =>)
      Move(in := #JOB_6_STEP_80, out1 => "Unit1.Em5.ControlNodes".GRnR_TransferPnP.sequence.status.nextStep)
   END_RUNG
   // the same network as SCL:
   #_w1 := ("Unit1.Em5.ControlNodes".GRnR_TransferPnP.sequence.status.currentStep = #JOB_6_STEP_50) AND "Unit1.Em5.ControlNodes".GRnR_TransferPnP.sequence.status.seqActive;
   "Unit1.Em5.ControlNodes".GRnR_TransferPnP."step".action1[650] := #_w1 AND NOT "Unit1.Em5.ControlNodes".cmTransferPnPRightClampOpenClose.monitoring.inHomePos;
   "Unit1.Em5.ControlNodes".GRnR_TransferPnP."step".transition1[650] := #_w1 AND "Unit1.Em5.ControlNodes".cmTransferPnPRightClampOpenClose.monitoring.inHomePos;
   #statTonTime[650].TON(IN := #_w1 AND "Unit1.Em5.ControlNodes".GRnR_TransferPnP."step".transition1[650],
                         PT := #delayTime);
   IF #statTonTime[650].Q THEN
       "Unit1.Em5.ControlNodes".GRnR_TransferPnP.sequence.status.nextStep := #JOB_6_STEP_80;
   END_IF;
END_REGION

REGION Network 19: Step[680] : Transfer PP Right Y-Axis Wait Pos
   RUNG wire#powerrail
      { S7_Templates := "SrcType := DInt" } EQ_Contact(in1 := "Unit1.Em5.ControlNodes".GRnR_TransferPnP.sequence.status.currentStep, in2 := #JOB_6_STEP_80)
      Contact( "Unit1.Em5.ControlNodes".GRnR_TransferPnP.sequence.status.seqActive )
      wire#w1
      I_Contact( "Unit1.Em5.ControlNodes".cm.softcam.transferPnPRightAxisY.pos00_wait.inPos )
      Coil( "Unit1.Em5.ControlNodes".GRnR_TransferPnP."step".action1[680] )
   END_RUNG
   RUNG wire#w1
      Contact( "Unit1.Em5.ControlNodes".cm.softcam.transferPnPRightAxisY.pos00_wait.inPos )
      Coil( "Unit1.Em5.ControlNodes".GRnR_TransferPnP."step".transition1[680] )
   END_RUNG
   RUNG wire#w1
      Contact( "Unit1.Em5.ControlNodes".GRnR_TransferPnP."step".transition1[680] )
      { S7_Templates := "time_type := Time" } #statTonTime[680].TON(pt := T#100ms, et =>)
      Move(in := #JOB_6_STEP_90, out1 => "Unit1.Em5.ControlNodes".GRnR_TransferPnP.sequence.status.nextStep)
   END_RUNG
   // the same network as SCL:
   #_w1 := ("Unit1.Em5.ControlNodes".GRnR_TransferPnP.sequence.status.currentStep = #JOB_6_STEP_80) AND "Unit1.Em5.ControlNodes".GRnR_TransferPnP.sequence.status.seqActive;
   "Unit1.Em5.ControlNodes".GRnR_TransferPnP."step".action1[680] := #_w1 AND NOT "Unit1.Em5.ControlNodes".cm.softcam.transferPnPRightAxisY.pos00_wait.inPos;
   "Unit1.Em5.ControlNodes".GRnR_TransferPnP."step".transition1[680] := #_w1 AND "Unit1.Em5.ControlNodes".cm.softcam.transferPnPRightAxisY.pos00_wait.inPos;
   #statTonTime[680].TON(IN := #_w1 AND "Unit1.Em5.ControlNodes".GRnR_TransferPnP."step".transition1[680],
                         PT := T#100ms);
   IF #statTonTime[680].Q THEN
       "Unit1.Em5.ControlNodes".GRnR_TransferPnP.sequence.status.nextStep := #JOB_6_STEP_90;
   END_IF;
END_REGION

REGION Network 20: Step[690] : JOB[6] Step End
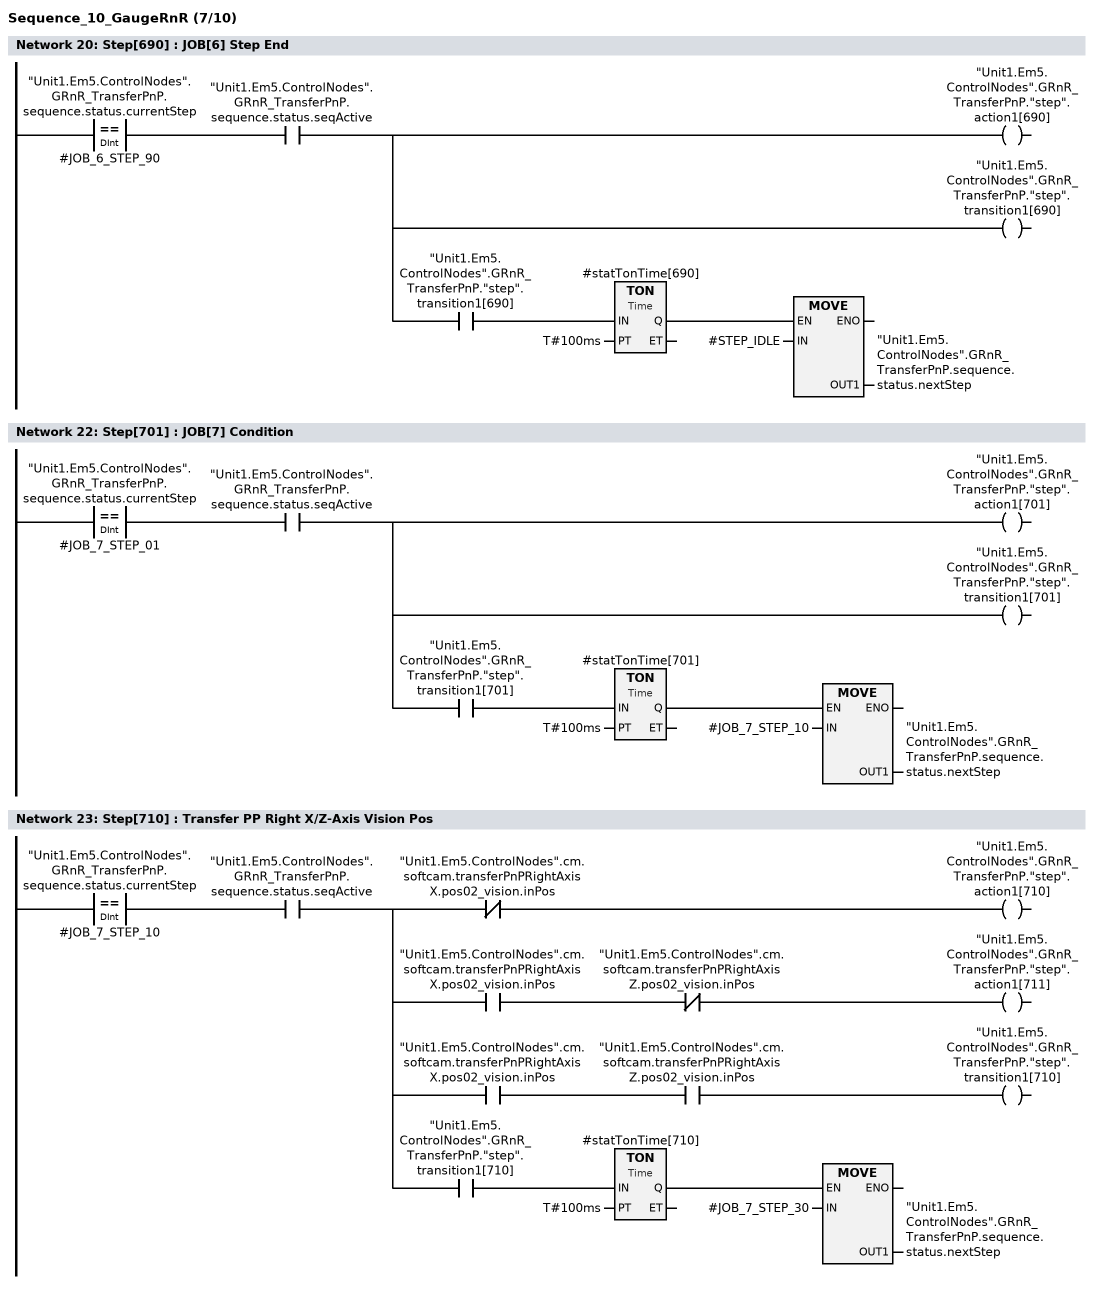
   RUNG wire#powerrail
      { S7_Templates := "SrcType := DInt" } EQ_Contact(in1 := "Unit1.Em5.ControlNodes".GRnR_TransferPnP.sequence.status.currentStep, in2 := #JOB_6_STEP_90)
      Contact( "Unit1.Em5.ControlNodes".GRnR_TransferPnP.sequence.status.seqActive )
      wire#w1
      Coil( "Unit1.Em5.ControlNodes".GRnR_TransferPnP."step".action1[690] )
   END_RUNG
   RUNG wire#w1
      Coil( "Unit1.Em5.ControlNodes".GRnR_TransferPnP."step".transition1[690] )
   END_RUNG
   RUNG wire#w1
      Contact( "Unit1.Em5.ControlNodes".GRnR_TransferPnP."step".transition1[690] )
      { S7_Templates := "time_type := Time" } #statTonTime[690].TON(pt := T#100ms, et =>)
      Move(in := #STEP_IDLE, out1 => "Unit1.Em5.ControlNodes".GRnR_TransferPnP.sequence.status.nextStep)
   END_RUNG
   // the same network as SCL:
   "Unit1.Em5.ControlNodes".GRnR_TransferPnP."step".action1[690] := ("Unit1.Em5.ControlNodes".GRnR_TransferPnP.sequence.status.currentStep = #JOB_6_STEP_90) AND "Unit1.Em5.ControlNodes".GRnR_TransferPnP.sequence.status.seqActive;
   "Unit1.Em5.ControlNodes".GRnR_TransferPnP."step".transition1[690] := ("Unit1.Em5.ControlNodes".GRnR_TransferPnP.sequence.status.currentStep = #JOB_6_STEP_90) AND "Unit1.Em5.ControlNodes".GRnR_TransferPnP.sequence.status.seqActive;
   #statTonTime[690].TON(IN := ("Unit1.Em5.ControlNodes".GRnR_TransferPnP.sequence.status.currentStep = #JOB_6_STEP_90) AND "Unit1.Em5.ControlNodes".GRnR_TransferPnP.sequence.status.seqActive AND "Unit1.Em5.ControlNodes".GRnR_TransferPnP."step".transition1[690],
                         PT := T#100ms);
   IF #statTonTime[690].Q THEN
       "Unit1.Em5.ControlNodes".GRnR_TransferPnP.sequence.status.nextStep := #STEP_IDLE;
   END_IF;
END_REGION

REGION Network 21: **************** JOB[7] VISION JR GET=R&R AUTO/TR RIGHT *****************
END_REGION

REGION Network 22: Step[701] : JOB[7] Condition
   RUNG wire#powerrail
      { S7_Templates := "SrcType := DInt" } EQ_Contact(in1 := "Unit1.Em5.ControlNodes".GRnR_TransferPnP.sequence.status.currentStep, in2 := #JOB_7_STEP_01)
      Contact( "Unit1.Em5.ControlNodes".GRnR_TransferPnP.sequence.status.seqActive )
      wire#w1
      Coil( "Unit1.Em5.ControlNodes".GRnR_TransferPnP."step".action1[701] )
   END_RUNG
   RUNG wire#w1
      Coil( "Unit1.Em5.ControlNodes".GRnR_TransferPnP."step".transition1[701] )
   END_RUNG
   RUNG wire#w1
      Contact( "Unit1.Em5.ControlNodes".GRnR_TransferPnP."step".transition1[701] )
      { S7_Templates := "time_type := Time" } #statTonTime[701].TON(pt := T#100ms, et =>)
      Move(in := #JOB_7_STEP_10, out1 => "Unit1.Em5.ControlNodes".GRnR_TransferPnP.sequence.status.nextStep)
   END_RUNG
   // the same network as SCL:
   "Unit1.Em5.ControlNodes".GRnR_TransferPnP."step".action1[701] := ("Unit1.Em5.ControlNodes".GRnR_TransferPnP.sequence.status.currentStep = #JOB_7_STEP_01) AND "Unit1.Em5.ControlNodes".GRnR_TransferPnP.sequence.status.seqActive;
   "Unit1.Em5.ControlNodes".GRnR_TransferPnP."step".transition1[701] := ("Unit1.Em5.ControlNodes".GRnR_TransferPnP.sequence.status.currentStep = #JOB_7_STEP_01) AND "Unit1.Em5.ControlNodes".GRnR_TransferPnP.sequence.status.seqActive;
   #statTonTime[701].TON(IN := ("Unit1.Em5.ControlNodes".GRnR_TransferPnP.sequence.status.currentStep = #JOB_7_STEP_01) AND "Unit1.Em5.ControlNodes".GRnR_TransferPnP.sequence.status.seqActive AND "Unit1.Em5.ControlNodes".GRnR_TransferPnP."step".transition1[701],
                         PT := T#100ms);
   IF #statTonTime[701].Q THEN
       "Unit1.Em5.ControlNodes".GRnR_TransferPnP.sequence.status.nextStep := #JOB_7_STEP_10;
   END_IF;
END_REGION

REGION Network 23: Step[710] : Transfer PP Right X/Z-Axis Vision Pos
   RUNG wire#powerrail
      { S7_Templates := "SrcType := DInt" } EQ_Contact(in1 := "Unit1.Em5.ControlNodes".GRnR_TransferPnP.sequence.status.currentStep, in2 := #JOB_7_STEP_10)
      Contact( "Unit1.Em5.ControlNodes".GRnR_TransferPnP.sequence.status.seqActive )
      wire#w1
      I_Contact( "Unit1.Em5.ControlNodes".cm.softcam.transferPnPRightAxisX.pos02_vision.inPos )
      Coil( "Unit1.Em5.ControlNodes".GRnR_TransferPnP."step".action1[710] )
   END_RUNG
   RUNG wire#w1
      Contact( "Unit1.Em5.ControlNodes".cm.softcam.transferPnPRightAxisX.pos02_vision.inPos )
      I_Contact( "Unit1.Em5.ControlNodes".cm.softcam.transferPnPRightAxisZ.pos02_vision.inPos )
      Coil( "Unit1.Em5.ControlNodes".GRnR_TransferPnP."step".action1[711] )
   END_RUNG
   RUNG wire#w1
      Contact( "Unit1.Em5.ControlNodes".cm.softcam.transferPnPRightAxisX.pos02_vision.inPos )
      Contact( "Unit1.Em5.ControlNodes".cm.softcam.transferPnPRightAxisZ.pos02_vision.inPos )
      Coil( "Unit1.Em5.ControlNodes".GRnR_TransferPnP."step".transition1[710] )
   END_RUNG
   RUNG wire#w1
      Contact( "Unit1.Em5.ControlNodes".GRnR_TransferPnP."step".transition1[710] )
      { S7_Templates := "time_type := Time" } #statTonTime[710].TON(pt := T#100ms, et =>)
      Move(in := #JOB_7_STEP_30, out1 => "Unit1.Em5.ControlNodes".GRnR_TransferPnP.sequence.status.nextStep)
   END_RUNG
   // the same network as SCL:
   #_w1 := ("Unit1.Em5.ControlNodes".GRnR_TransferPnP.sequence.status.currentStep = #JOB_7_STEP_10) AND "Unit1.Em5.ControlNodes".GRnR_TransferPnP.sequence.status.seqActive;
   "Unit1.Em5.ControlNodes".GRnR_TransferPnP."step".action1[710] := #_w1 AND NOT "Unit1.Em5.ControlNodes".cm.softcam.transferPnPRightAxisX.pos02_vision.inPos;
   "Unit1.Em5.ControlNodes".GRnR_TransferPnP."step".action1[711] := #_w1 AND "Unit1.Em5.ControlNodes".cm.softcam.transferPnPRightAxisX.pos02_vision.inPos AND NOT "Unit1.Em5.ControlNodes".cm.softcam.transferPnPRightAxisZ.pos02_vision.inPos;
   "Unit1.Em5.ControlNodes".GRnR_TransferPnP."step".transition1[710] := #_w1 AND "Unit1.Em5.ControlNodes".cm.softcam.transferPnPRightAxisX.pos02_vision.inPos AND "Unit1.Em5.ControlNodes".cm.softcam.transferPnPRightAxisZ.pos02_vision.inPos;
   #statTonTime[710].TON(IN := #_w1 AND "Unit1.Em5.ControlNodes".GRnR_TransferPnP."step".transition1[710],
                         PT := T#100ms);
   IF #statTonTime[710].Q THEN
       "Unit1.Em5.ControlNodes".GRnR_TransferPnP.sequence.status.nextStep := #JOB_7_STEP_30;
   END_IF;
END_REGION

REGION Network 24: Step[730] : Transfer PP Right Y-Axis Vision Pos
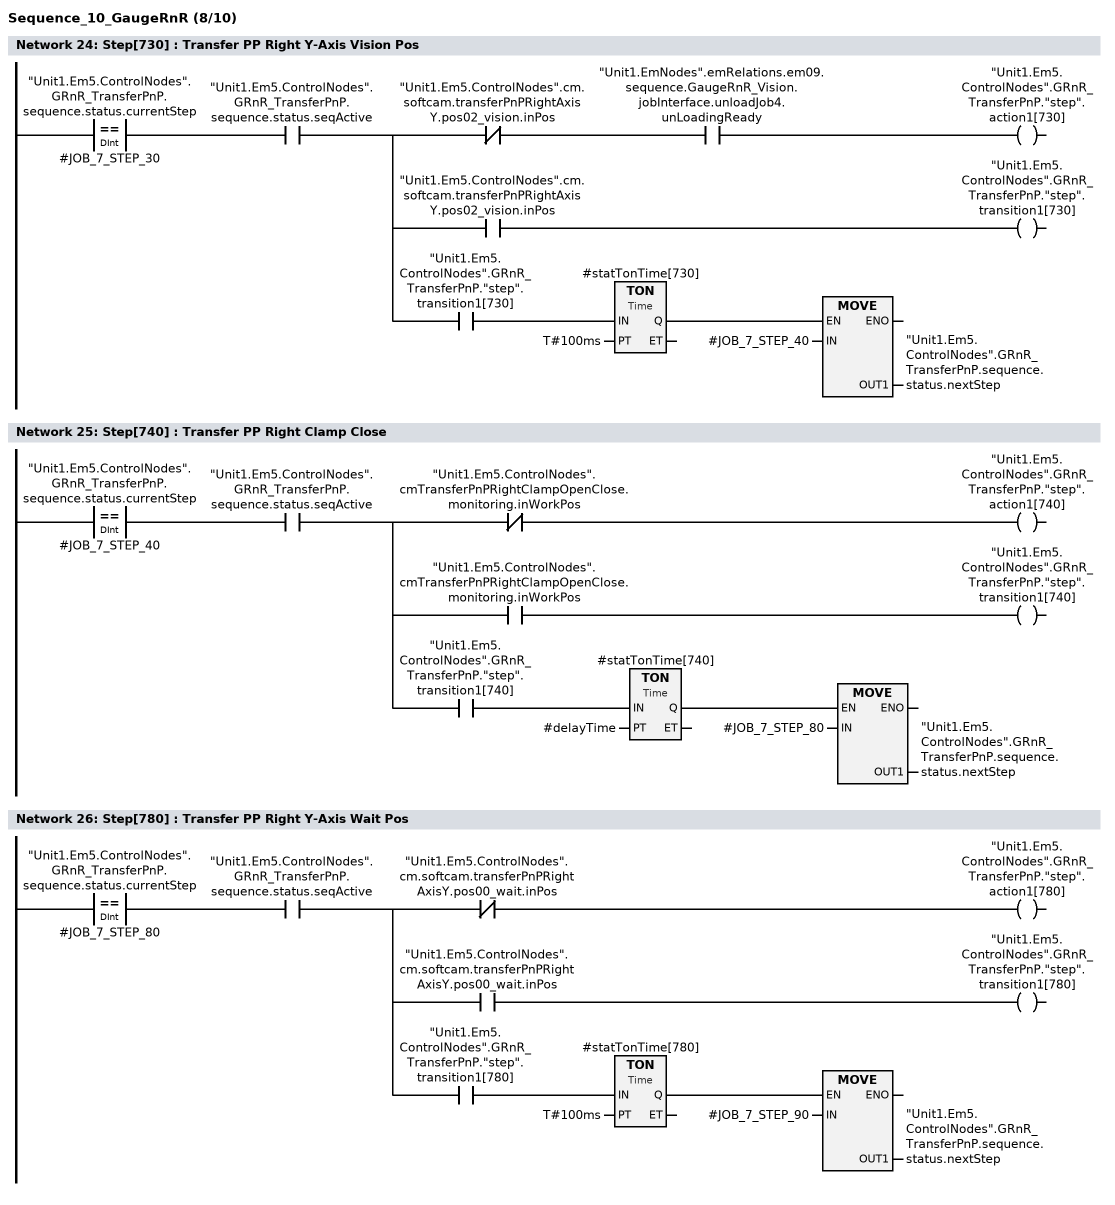
   RUNG wire#powerrail
      { S7_Templates := "SrcType := DInt" } EQ_Contact(in1 := "Unit1.Em5.ControlNodes".GRnR_TransferPnP.sequence.status.currentStep, in2 := #JOB_7_STEP_30)
      Contact( "Unit1.Em5.ControlNodes".GRnR_TransferPnP.sequence.status.seqActive )
      wire#w1
      I_Contact( "Unit1.Em5.ControlNodes".cm.softcam.transferPnPRightAxisY.pos02_vision.inPos )
      Contact( "Unit1.EmNodes".emRelations.em09.sequence.GaugeRnR_Vision.jobInterface.unloadJob4.unLoadingReady )
      Coil( "Unit1.Em5.ControlNodes".GRnR_TransferPnP."step".action1[730] )
   END_RUNG
   RUNG wire#w1
      Contact( "Unit1.Em5.ControlNodes".cm.softcam.transferPnPRightAxisY.pos02_vision.inPos )
      Coil( "Unit1.Em5.ControlNodes".GRnR_TransferPnP."step".transition1[730] )
   END_RUNG
   RUNG wire#w1
      Contact( "Unit1.Em5.ControlNodes".GRnR_TransferPnP."step".transition1[730] )
      { S7_Templates := "time_type := Time" } #statTonTime[730].TON(pt := T#100ms, et =>)
      Move(in := #JOB_7_STEP_40, out1 => "Unit1.Em5.ControlNodes".GRnR_TransferPnP.sequence.status.nextStep)
   END_RUNG
   // the same network as SCL:
   #_w1 := ("Unit1.Em5.ControlNodes".GRnR_TransferPnP.sequence.status.currentStep = #JOB_7_STEP_30) AND "Unit1.Em5.ControlNodes".GRnR_TransferPnP.sequence.status.seqActive;
   "Unit1.Em5.ControlNodes".GRnR_TransferPnP."step".action1[730] := #_w1 AND NOT "Unit1.Em5.ControlNodes".cm.softcam.transferPnPRightAxisY.pos02_vision.inPos AND "Unit1.EmNodes".emRelations.em09.sequence.GaugeRnR_Vision.jobInterface.unloadJob4.unLoadingReady;
   "Unit1.Em5.ControlNodes".GRnR_TransferPnP."step".transition1[730] := #_w1 AND "Unit1.Em5.ControlNodes".cm.softcam.transferPnPRightAxisY.pos02_vision.inPos;
   #statTonTime[730].TON(IN := #_w1 AND "Unit1.Em5.ControlNodes".GRnR_TransferPnP."step".transition1[730],
                         PT := T#100ms);
   IF #statTonTime[730].Q THEN
       "Unit1.Em5.ControlNodes".GRnR_TransferPnP.sequence.status.nextStep := #JOB_7_STEP_40;
   END_IF;
END_REGION

REGION Network 25: Step[740] : Transfer PP Right Clamp Close
   RUNG wire#powerrail
      { S7_Templates := "SrcType := DInt" } EQ_Contact(in1 := "Unit1.Em5.ControlNodes".GRnR_TransferPnP.sequence.status.currentStep, in2 := #JOB_7_STEP_40)
      Contact( "Unit1.Em5.ControlNodes".GRnR_TransferPnP.sequence.status.seqActive )
      wire#w1
      I_Contact( "Unit1.Em5.ControlNodes".cmTransferPnPRightClampOpenClose.monitoring.inWorkPos )
      Coil( "Unit1.Em5.ControlNodes".GRnR_TransferPnP."step".action1[740] )
   END_RUNG
   RUNG wire#w1
      Contact( "Unit1.Em5.ControlNodes".cmTransferPnPRightClampOpenClose.monitoring.inWorkPos )
      Coil( "Unit1.Em5.ControlNodes".GRnR_TransferPnP."step".transition1[740] )
   END_RUNG
   RUNG wire#w1
      Contact( "Unit1.Em5.ControlNodes".GRnR_TransferPnP."step".transition1[740] )
      { S7_Templates := "time_type := Time" } #statTonTime[740].TON(pt := #delayTime, et =>)
      Move(in := #JOB_7_STEP_80, out1 => "Unit1.Em5.ControlNodes".GRnR_TransferPnP.sequence.status.nextStep)
   END_RUNG
   // the same network as SCL:
   #_w1 := ("Unit1.Em5.ControlNodes".GRnR_TransferPnP.sequence.status.currentStep = #JOB_7_STEP_40) AND "Unit1.Em5.ControlNodes".GRnR_TransferPnP.sequence.status.seqActive;
   "Unit1.Em5.ControlNodes".GRnR_TransferPnP."step".action1[740] := #_w1 AND NOT "Unit1.Em5.ControlNodes".cmTransferPnPRightClampOpenClose.monitoring.inWorkPos;
   "Unit1.Em5.ControlNodes".GRnR_TransferPnP."step".transition1[740] := #_w1 AND "Unit1.Em5.ControlNodes".cmTransferPnPRightClampOpenClose.monitoring.inWorkPos;
   #statTonTime[740].TON(IN := #_w1 AND "Unit1.Em5.ControlNodes".GRnR_TransferPnP."step".transition1[740],
                         PT := #delayTime);
   IF #statTonTime[740].Q THEN
       "Unit1.Em5.ControlNodes".GRnR_TransferPnP.sequence.status.nextStep := #JOB_7_STEP_80;
   END_IF;
END_REGION

REGION Network 26: Step[780] : Transfer PP Right Y-Axis Wait Pos
   RUNG wire#powerrail
      { S7_Templates := "SrcType := DInt" } EQ_Contact(in1 := "Unit1.Em5.ControlNodes".GRnR_TransferPnP.sequence.status.currentStep, in2 := #JOB_7_STEP_80)
      Contact( "Unit1.Em5.ControlNodes".GRnR_TransferPnP.sequence.status.seqActive )
      wire#w1
      I_Contact( "Unit1.Em5.ControlNodes".cm.softcam.transferPnPRightAxisY.pos00_wait.inPos )
      Coil( "Unit1.Em5.ControlNodes".GRnR_TransferPnP."step".action1[780] )
   END_RUNG
   RUNG wire#w1
      Contact( "Unit1.Em5.ControlNodes".cm.softcam.transferPnPRightAxisY.pos00_wait.inPos )
      Coil( "Unit1.Em5.ControlNodes".GRnR_TransferPnP."step".transition1[780] )
   END_RUNG
   RUNG wire#w1
      Contact( "Unit1.Em5.ControlNodes".GRnR_TransferPnP."step".transition1[780] )
      { S7_Templates := "time_type := Time" } #statTonTime[780].TON(pt := T#100ms, et =>)
      Move(in := #JOB_7_STEP_90, out1 => "Unit1.Em5.ControlNodes".GRnR_TransferPnP.sequence.status.nextStep)
   END_RUNG
   // the same network as SCL:
   #_w1 := ("Unit1.Em5.ControlNodes".GRnR_TransferPnP.sequence.status.currentStep = #JOB_7_STEP_80) AND "Unit1.Em5.ControlNodes".GRnR_TransferPnP.sequence.status.seqActive;
   "Unit1.Em5.ControlNodes".GRnR_TransferPnP."step".action1[780] := #_w1 AND NOT "Unit1.Em5.ControlNodes".cm.softcam.transferPnPRightAxisY.pos00_wait.inPos;
   "Unit1.Em5.ControlNodes".GRnR_TransferPnP."step".transition1[780] := #_w1 AND "Unit1.Em5.ControlNodes".cm.softcam.transferPnPRightAxisY.pos00_wait.inPos;
   #statTonTime[780].TON(IN := #_w1 AND "Unit1.Em5.ControlNodes".GRnR_TransferPnP."step".transition1[780],
                         PT := T#100ms);
   IF #statTonTime[780].Q THEN
       "Unit1.Em5.ControlNodes".GRnR_TransferPnP.sequence.status.nextStep := #JOB_7_STEP_90;
   END_IF;
END_REGION

REGION Network 27: Step[790] : JOB[7] Step End
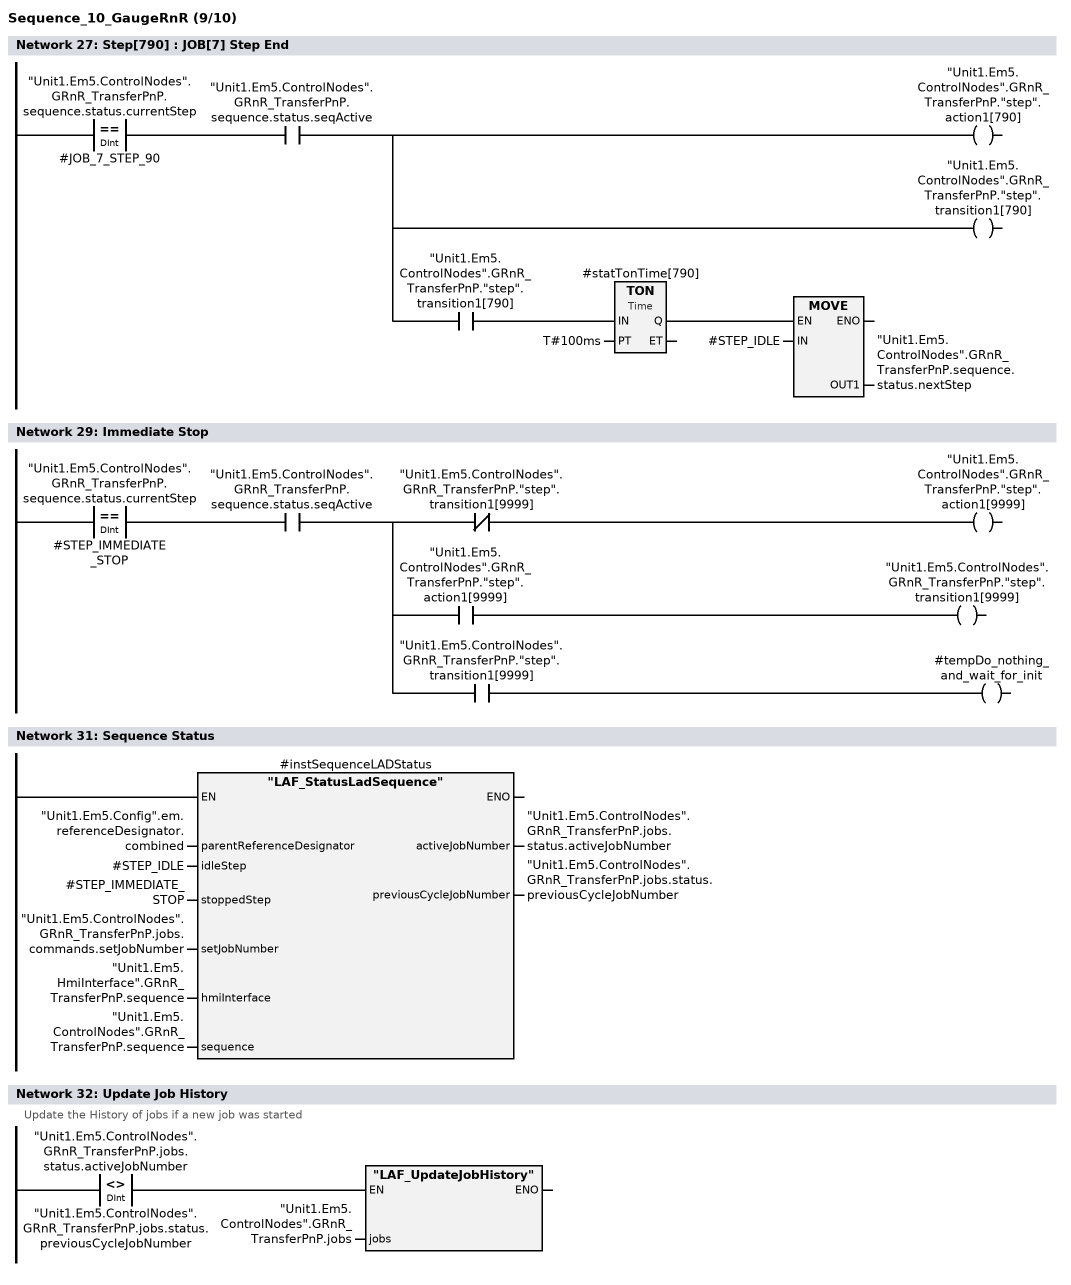
   RUNG wire#powerrail
      { S7_Templates := "SrcType := DInt" } EQ_Contact(in1 := "Unit1.Em5.ControlNodes".GRnR_TransferPnP.sequence.status.currentStep, in2 := #JOB_7_STEP_90)
      Contact( "Unit1.Em5.ControlNodes".GRnR_TransferPnP.sequence.status.seqActive )
      wire#w1
      Coil( "Unit1.Em5.ControlNodes".GRnR_TransferPnP."step".action1[790] )
   END_RUNG
   RUNG wire#w1
      Coil( "Unit1.Em5.ControlNodes".GRnR_TransferPnP."step".transition1[790] )
   END_RUNG
   RUNG wire#w1
      Contact( "Unit1.Em5.ControlNodes".GRnR_TransferPnP."step".transition1[790] )
      { S7_Templates := "time_type := Time" } #statTonTime[790].TON(pt := T#100ms, et =>)
      Move(in := #STEP_IDLE, out1 => "Unit1.Em5.ControlNodes".GRnR_TransferPnP.sequence.status.nextStep)
   END_RUNG
   // the same network as SCL:
   "Unit1.Em5.ControlNodes".GRnR_TransferPnP."step".action1[790] := ("Unit1.Em5.ControlNodes".GRnR_TransferPnP.sequence.status.currentStep = #JOB_7_STEP_90) AND "Unit1.Em5.ControlNodes".GRnR_TransferPnP.sequence.status.seqActive;
   "Unit1.Em5.ControlNodes".GRnR_TransferPnP."step".transition1[790] := ("Unit1.Em5.ControlNodes".GRnR_TransferPnP.sequence.status.currentStep = #JOB_7_STEP_90) AND "Unit1.Em5.ControlNodes".GRnR_TransferPnP.sequence.status.seqActive;
   #statTonTime[790].TON(IN := ("Unit1.Em5.ControlNodes".GRnR_TransferPnP.sequence.status.currentStep = #JOB_7_STEP_90) AND "Unit1.Em5.ControlNodes".GRnR_TransferPnP.sequence.status.seqActive AND "Unit1.Em5.ControlNodes".GRnR_TransferPnP."step".transition1[790],
                         PT := T#100ms);
   IF #statTonTime[790].Q THEN
       "Unit1.Em5.ControlNodes".GRnR_TransferPnP.sequence.status.nextStep := #STEP_IDLE;
   END_IF;
END_REGION

REGION Network 28: ******************** IMMEDIATE STOP *********************
END_REGION

REGION Network 29: Immediate Stop
   RUNG wire#powerrail
      { S7_Templates := "SrcType := DInt" } EQ_Contact(in1 := "Unit1.Em5.ControlNodes".GRnR_TransferPnP.sequence.status.currentStep, in2 := #STEP_IMMEDIATE_STOP)
      Contact( "Unit1.Em5.ControlNodes".GRnR_TransferPnP.sequence.status.seqActive )
      wire#w1
      I_Contact( "Unit1.Em5.ControlNodes".GRnR_TransferPnP."step".transition1[9999] )
      Coil( "Unit1.Em5.ControlNodes".GRnR_TransferPnP."step".action1[9999] )
   END_RUNG
   RUNG wire#w1
      Contact( "Unit1.Em5.ControlNodes".GRnR_TransferPnP."step".action1[9999] )
      Coil( "Unit1.Em5.ControlNodes".GRnR_TransferPnP."step".transition1[9999] )
   END_RUNG
   RUNG wire#w1
      Contact( "Unit1.Em5.ControlNodes".GRnR_TransferPnP."step".transition1[9999] )
      Coil( #tempDo_nothing_and_wait_for_init )
   END_RUNG
   // the same network as SCL:
   #_w1 := ("Unit1.Em5.ControlNodes".GRnR_TransferPnP.sequence.status.currentStep = #STEP_IMMEDIATE_STOP) AND "Unit1.Em5.ControlNodes".GRnR_TransferPnP.sequence.status.seqActive;
   "Unit1.Em5.ControlNodes".GRnR_TransferPnP."step".action1[9999] := #_w1 AND NOT "Unit1.Em5.ControlNodes".GRnR_TransferPnP."step".transition1[9999];
   "Unit1.Em5.ControlNodes".GRnR_TransferPnP."step".transition1[9999] := #_w1 AND "Unit1.Em5.ControlNodes".GRnR_TransferPnP."step".action1[9999];
   #tempDo_nothing_and_wait_for_init := #_w1 AND "Unit1.Em5.ControlNodes".GRnR_TransferPnP."step".transition1[9999];
END_REGION

REGION Network 30: ********************** STATUS **************************
END_REGION

REGION Network 31: Sequence Status
   RUNG wire#powerrail
      #instSequenceLADStatus(parentReferenceDesignator := "Unit1.Em5.Config".em.referenceDesignator.combined, idleStep := #STEP_IDLE, stoppedStep := #STEP_IMMEDIATE_STOP, setJobNumber := "Unit1.Em5.ControlNodes".GRnR_TransferPnP.jobs.commands.setJobNumber, hmiInterface := "Unit1.Em5.HmiInterface".GRnR_TransferPnP.sequence, sequence := "Unit1.Em5.ControlNodes".GRnR_TransferPnP.sequence, activeJobNumber => "Unit1.Em5.ControlNodes".GRnR_TransferPnP.jobs.status.activeJobNumber, previousCycleJobNumber => "Unit1.Em5.ControlNodes".GRnR_TransferPnP.jobs.status.previousCycleJobNumber)
   END_RUNG
   // the same network as SCL:
   #instSequenceLADStatus(parentReferenceDesignator := "Unit1.Em5.Config".em.referenceDesignator.combined,   // "LAF_StatusLadSequence"
                          idleStep := #STEP_IDLE,
                          stoppedStep := #STEP_IMMEDIATE_STOP,
                          setJobNumber := "Unit1.Em5.ControlNodes".GRnR_TransferPnP.jobs.commands.setJobNumber,
                          hmiInterface := "Unit1.Em5.HmiInterface".GRnR_TransferPnP.sequence,
                          sequence := "Unit1.Em5.ControlNodes".GRnR_TransferPnP.sequence,
                          activeJobNumber => "Unit1.Em5.ControlNodes".GRnR_TransferPnP.jobs.status.activeJobNumber,
                          previousCycleJobNumber => "Unit1.Em5.ControlNodes".GRnR_TransferPnP.jobs.status.previousCycleJobNumber);
END_REGION

REGION Network 32: Update Job History
   // Update the History of jobs if a new job was started
   RUNG wire#powerrail
      { S7_Templates := "SrcType := DInt" } NE_Contact(in1 := "Unit1.Em5.ControlNodes".GRnR_TransferPnP.jobs.status.activeJobNumber, in2 := "Unit1.Em5.ControlNodes".GRnR_TransferPnP.jobs.status.previousCycleJobNumber)
      "LAF_UpdateJobHistory"(jobs := "Unit1.Em5.ControlNodes".GRnR_TransferPnP.jobs)
   END_RUNG
   // the same network as SCL:
   IF "Unit1.Em5.ControlNodes".GRnR_TransferPnP.jobs.status.activeJobNumber <> "Unit1.Em5.ControlNodes".GRnR_TransferPnP.jobs.status.previousCycleJobNumber THEN
       "LAF_UpdateJobHistory"(jobs := "Unit1.Em5.ControlNodes".GRnR_TransferPnP.jobs);
   END_IF;
END_REGION

REGION Network 33: Output Steps As String
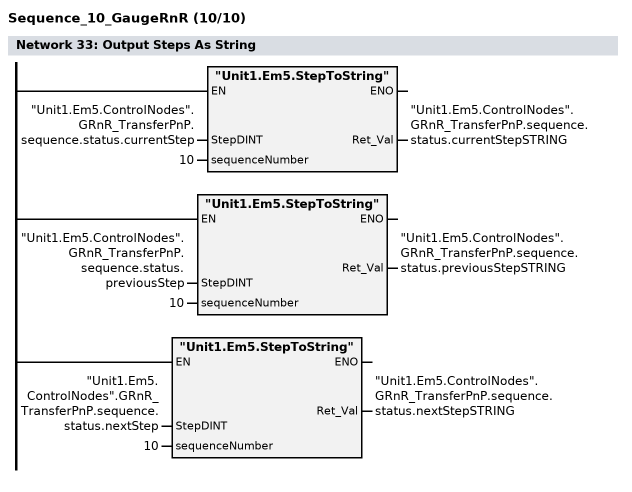
   RUNG wire#powerrail
      "Unit1.Em5.StepToString"(StepDINT := "Unit1.Em5.ControlNodes".GRnR_TransferPnP.sequence.status.currentStep, sequenceNumber := 10, Ret_Val => "Unit1.Em5.ControlNodes".GRnR_TransferPnP.sequence.status.currentStepSTRING)
   END_RUNG
   RUNG wire#powerrail
      "Unit1.Em5.StepToString"(StepDINT := "Unit1.Em5.ControlNodes".GRnR_TransferPnP.sequence.status.previousStep, sequenceNumber := 10, Ret_Val => "Unit1.Em5.ControlNodes".GRnR_TransferPnP.sequence.status.previousStepSTRING)
   END_RUNG
   RUNG wire#powerrail
      "Unit1.Em5.StepToString"(StepDINT := "Unit1.Em5.ControlNodes".GRnR_TransferPnP.sequence.status.nextStep, sequenceNumber := 10, Ret_Val => "Unit1.Em5.ControlNodes".GRnR_TransferPnP.sequence.status.nextStepSTRING)
   END_RUNG
   // the same network as SCL:
   "Unit1.Em5.ControlNodes".GRnR_TransferPnP.sequence.status.currentStepSTRING := "Unit1.Em5.StepToString"(StepDINT := "Unit1.Em5.ControlNodes".GRnR_TransferPnP.sequence.status.currentStep,
                           sequenceNumber := 10);
   "Unit1.Em5.ControlNodes".GRnR_TransferPnP.sequence.status.previousStepSTRING := "Unit1.Em5.StepToString"(StepDINT := "Unit1.Em5.ControlNodes".GRnR_TransferPnP.sequence.status.previousStep,
                           sequenceNumber := 10);
   "Unit1.Em5.ControlNodes".GRnR_TransferPnP.sequence.status.nextStepSTRING := "Unit1.Em5.StepToString"(StepDINT := "Unit1.Em5.ControlNodes".GRnR_TransferPnP.sequence.status.nextStep,
                           sequenceNumber := 10);
END_REGION
END_FUNCTION_BLOCK
